LIN {X 0,Y 205.267,Z 502.12,A -85,B 0,C 180,E1 -21304.12,E2 -21304.12} C_VEL
LIN {X 0,Y 202.295,Z 509.063,A -85,B 0,C 180,E1 -21307.536,E2 -21307.536} C_VEL
LIN {X 0,Y 199.763,Z 515.879,A -85,B 0,C 180,E1 -21311.788,E2 -21311.788} C_VEL
LIN {X 0,Y 198.325,Z 520.575,A -85,B 0,C 180,E1 -21315.64,E2 -21315.64} C_VEL
LIN {X 0,Y 197.677,Z 524.301,A -85,B 0,C 180,E1 -21319.763,E2 -21319.763} C_VEL
LIN {X 0,Y 197.879,Z 526.838,A -85,B 0,C 180,E1 -21323.967,E2 -21323.967} C_VEL
LIN {X 0,Y 198.163,Z 528.073,A -85,B 0,C 180,E1 -21327.97,E2 -21327.97} C_VEL
LIN {X 0,Y 198.486,Z 528.261,A -85,B 0,C 180,E1 -21330.003,E2 -21330.003} C_VEL
LIN {X 0,Y 198.017,Z 527.58,A -85,B 0,C 180,E1 -21334.073,E2 -21334.073} C_VEL
LIN {X 0,Y 197.928,Z 526.77,A -85,B 0,C 180,E1 -21336.164,E2 -21336.164} C_VEL
LIN {X 0,Y 197.717,Z 524.267,A -85,B 0,C 180,E1 -21340.24,E2 -21340.24} C_VEL
LIN {X 0,Y 198.347,Z 520.514,A -85,B 0,C 180,E1 -21344.363,E2 -21344.363} C_VEL
LIN {X 0,Y 199.847,Z 515.452,A -85,B 0,C 180,E1 -21348.454,E2 -21348.454} C_VEL
LIN {X 0,Y 202.319,Z 508.963,A -85,B 0,C 180,E1 -21352.467,E2 -21352.467} C_VEL
LIN {X 0,Y 205.735,Z 500.856,A -85,B 0,C 180,E1 -21356.367,E2 -21356.367} C_VEL
LIN {X 0,Y 208.882,Z 493.891,A -85,B 0,C 180,E1 -21359.202,E2 -21359.202} C_VEL
LIN {X 0,Y 214.362,Z 488.856,A -85,B 0,C 180,E1 -21362.752,E2 -21362.752} C_VEL
LIN {X 0,Y 222.751,Z 481.086,A -85,B 0,C 180,E1 -21366.834,E2 -21366.834} C_VEL
LIN {X 0,Y 228.645,Z 475.569,A -85,B 0,C 180,E1 -21369.061,E2 -21369.061} C_VEL
LIN {X 0,Y 239.611,Z 464.861,A -85,B 0,C 180,E1 -21372.426,E2 -21372.426} C_VEL
LIN {X 0,Y 250.645,Z 453.222,A -85,B 0,C 180,E1 -21375.075,E2 -21375.075} C_VEL
LIN {X 0,Y 261.321,Z 440.945,A -85,B 0,C 180,E1 -21377.129,E2 -21377.129} C_VEL
LIN {X 0,Y 269.925,Z 430.113,A -85,B 0,C 180,E1 -21378.468,E2 -21378.468} C_VEL
LIN {X 0,Y 275.364,Z 422.771,A -85,B 0,C 180,E1 -21379.23,E2 -21379.23} C_VEL
LIN {X 0,Y 276.293,Z 421.354,A -85,B 0,C 180,E1 -21379.579,E2 -21379.579} C_VEL
LIN {X 0,Y 267.377,Z 431.541,A -85,B 0,C 180,E1 -21381.372,E2 -21381.372} C_VEL
LIN {X 0,Y 257.679,Z 441.222,A -85,B 0,C 180,E1 -21383.615,E2 -21383.615} C_VEL
LIN {X 0,Y 249.699,Z 448.11,A -85,B 0,C 180,E1 -21385.742,E2 -21385.742} C_VEL
LIN {X 0,Y 241.223,Z 454.408,A -85,B 0,C 180,E1 -21388.37,E2 -21388.37} C_VEL
LIN {X 0,Y 233.351,Z 459.281,A -85,B 0,C 180,E1 -21391.192,E2 -21391.192} C_VEL
LIN {X 0,Y 226.141,Z 462.776,A -85,B 0,C 180,E1 -21394.209,E2 -21394.209} C_VEL
LIN {X 0,Y 219.797,Z 464.844,A -85,B 0,C 180,E1 -21397.437,E2 -21397.437} C_VEL
LIN {X 0,Y 214.14,Z 465.558,A -85,B 0,C 180,E1 -21400.841,E2 -21400.841} C_VEL
LIN {X 0,Y 209.476,Z 464.862,A -85,B 0,C 180,E1 -21404.431,E2 -21404.431} C_VEL
LIN {X 0,Y 205.6,Z 462.774,A -85,B 0,C 180,E1 -21408.165,E2 -21408.165} C_VEL
LIN {X 0,Y 202.968,Z 459.202,A -85,B 0,C 180,E1 -21412.039,E2 -21412.039} C_VEL
LIN {X 0,Y 200.986,Z 454.078,A -85,B 0,C 180,E1 -21415.99,E2 -21415.99} C_VEL
LIN {X 0,Y 199.711,Z 447.24,A -85,B 0,C 180,E1 -21420,E2 -21420} C_VEL
LIN {X 0,Y 199.428,Z 440.84,A -85,B 0,C 180,E1 -21423.03,E2 -21423.03} C_VEL
LIN {X 0,Y 199.398,Z 433.173,A -85,B 0,C 180,E1 -21426.07,E2 -21426.07} C_VEL
LIN {X 0,Y 199.905,Z 424.141,A -85,B 0,C 180,E1 -21429.076,E2 -21429.076} C_VEL
LIN {X 0,Y 200.647,Z 413.012,A -85,B 0,C 180,E1 -21432.132,E2 -21432.132} C_VEL
LIN {X 0,Y 201.556,Z 400.828,A -85,B 0,C 180,E1 -21434.902,E2 -21434.902} C_VEL
LIN {X 0,Y 202.642,Z 387.299,A -85,B 0,C 180,E1 -21437.406,E2 -21437.406} C_VEL
LIN {X 0,Y 203.727,Z 374.15,A -85,B 0,C 180,E1 -21439.393,E2 -21439.393} C_VEL
LIN {X 0,Y 204.695,Z 359.774,A -85,B 0,C 180,E1 -21441.132,E2 -21441.132} C_VEL
LIN {X 0,Y 205.639,Z 343.824,A -85,B 0,C 180,E1 -21442.623,E2 -21442.623} C_VEL
LIN {X 0,Y 206.657,Z 321.429,A -85,B 0,C 180,E1 -21444.086,E2 -21444.086} C_VEL
LIN {X 0,Y 211.562,Z 242.2,A -85,B 0,C 180,E1 -21448.698,E2 -21448.698} C_VEL
LIN {X 0,Y 211.534,Z 241.628,A -85,B 0,C 180,E1 -21448.781,E2 -21448.781} C_VEL
LIN {X 0,Y 213.23,Z 241.827,A -85,B 0,C 180,E1 -21449.63,E2 -21449.63} C_VEL
LIN {X 0,Y 214.627,Z 239.56,A -85,B 0,C 180,E1 -21450.143,E2 -21450.143} C_VEL
LIN {X 0,Y 216.77,Z 233.61,A -85,B 0,C 180,E1 -21450.741,E2 -21450.741} C_VEL
LIN {X 0,Y 218.364,Z 227.891,A -85,B 0,C 180,E1 -21451.09,E2 -21451.09} C_VEL
LIN {X 0,Y 220.497,Z 225.426,A -85,B 0,C 180,E1 -21451.864,E2 -21451.864} C_VEL
LIN {X 0,Y 222.215,Z 222.209,A -85,B 0,C 180,E1 -21452.39,E2 -21452.39} C_VEL
LIN {X 0,Y 224.392,Z 221.596,A -85,B 0,C 180,E1 -21453.237,E2 -21453.237} C_VEL
LIN {X 0,Y 228.278,Z 221.524,A -85,B 0,C 180,E1 -21454.72,E2 -21454.72} C_VEL
LIN {X 0,Y 231.326,Z 221.102,A -85,B 0,C 180,E1 -21455.792,E2 -21455.792} C_VEL
LIN {X 0,Y 232.183,Z 221.454,A -85,B 0,C 180,E1 -21456.108,E2 -21456.108} C_VEL
LIN {X 0,Y 237.875,Z 230.482,A -85,B 0,C 180,E1 -21458.416,E2 -21458.416} C_VEL
LIN {X 0,Y 244.244,Z 241.683,A -85,B 0,C 180,E1 -21460.797,E2 -21460.797} C_VEL
LIN {X 0,Y 250.045,Z 253.287,A -85,B 0,C 180,E1 -21462.827,E2 -21462.827} C_VEL
LIN {X 0,Y 243.977,Z 351.523,A -85,B 0,C 180,E1 -21465.471,E2 -21465.471} C_VEL
LIN {X 0,Y 242.422,Z 366.589,A -85,B 0,C 180,E1 -21466.149,E2 -21466.149} C_VEL
LIN {X 0,Y 240.345,Z 380.819,A -85,B 0,C 180,E1 -21467.092,E2 -21467.092} C_VEL
LIN {X 0,Y 237.764,Z 394.532,A -85,B 0,C 180,E1 -21468.31,E2 -21468.31} C_VEL
LIN {X 0,Y 234.321,Z 408.371,A -85,B 0,C 180,E1 -21469.843,E2 -21469.843} C_VEL
LIN {X 0,Y 230.62,Z 420.997,A -85,B 0,C 180,E1 -21471.615,E2 -21471.615} C_VEL
LIN {X 0,Y 226.485,Z 432.68,A -85,B 0,C 180,E1 -21473.595,E2 -21473.595} C_VEL
LIN {X 0,Y 222.424,Z 443.47,A -85,B 0,C 180,E1 -21475.883,E2 -21475.883} C_VEL
LIN {X 0,Y 218.441,Z 453.372,A -85,B 0,C 180,E1 -21478.476,E2 -21478.476} C_VEL
LIN {X 0,Y 213.958,Z 463.052,A -85,B 0,C 180,E1 -21481.554,E2 -21481.554} C_VEL
LIN {X 0,Y 209.892,Z 471.448,A -85,B 0,C 180,E1 -21484.916,E2 -21484.916} C_VEL
LIN {X 0,Y 206.815,Z 477.669,A -85,B 0,C 180,E1 -21488.047,E2 -21488.047} C_VEL
LIN {X 0,Y 203.821,Z 483.766,A -85,B 0,C 180,E1 -21491.918,E2 -21491.918} C_VEL
LIN {X 0,Y 201.497,Z 488.471,A -85,B 0,C 180,E1 -21495.866,E2 -21495.866} C_VEL
LIN {X 0,Y 199.865,Z 491.947,A -85,B 0,C 180,E1 -21499.928,E2 -21499.928} C_VEL
LIN {X 0,Y 198.859,Z 494.17,A -85,B 0,C 180,E1 -21503.911,E2 -21503.911} C_VEL
LIN {X 0,Y 198.504,Z 495.303,A -85,B 0,C 180,E1 -21507.968,E2 -21507.968} C_VEL
LIN {X 0,Y 198.503,Z 495.314,A -85,B 0,C 180,E1 -21512.026,E2 -21512.026} C_VEL
LIN {X 0,Y 198.844,Z 494.224,A -85,B 0,C 180,E1 -21516.084,E2 -21516.084} C_VEL
LIN {X 0,Y 199.896,Z 492.006,A -85,B 0,C 180,E1 -21520.122,E2 -21520.122} C_VEL
LIN {X 0,Y 201.475,Z 488.625,A -85,B 0,C 180,E1 -21524.131,E2 -21524.131} C_VEL
LIN {X 0,Y 203.746,Z 483.977,A -85,B 0,C 180,E1 -21528.083,E2 -21528.083} C_VEL
LIN {X 0,Y 206.75,Z 477.926,A -85,B 0,C 180,E1 -21531.955,E2 -21531.955} C_VEL
LIN {X 0,Y 210.505,Z 470.295,A -85,B 0,C 180,E1 -21535.72,E2 -21535.72} C_VEL
LIN {X 0,Y 214.482,Z 462.127,A -85,B 0,C 180,E1 -21538.899,E2 -21538.899} C_VEL
LIN {X 0,Y 218.318,Z 453.818,A -85,B 0,C 180,E1 -21541.538,E2 -21541.538} C_VEL
LIN {X 0,Y 223.004,Z 442.178,A -85,B 0,C 180,E1 -21544.557,E2 -21544.557} C_VEL
LIN {X 0,Y 227.205,Z 431.186,A -85,B 0,C 180,E1 -21546.818,E2 -21546.818} C_VEL
LIN {X 0,Y 231.291,Z 419.223,A -85,B 0,C 180,E1 -21548.804,E2 -21548.804} C_VEL
LIN {X 0,Y 235.067,Z 406.182,A -85,B 0,C 180,E1 -21550.559,E2 -21550.559} C_VEL
LIN {X 0,Y 238.502,Z 391.783,A -85,B 0,C 180,E1 -21552.093,E2 -21552.093} C_VEL
LIN {X 0,Y 241.052,Z 377.556,A -85,B 0,C 180,E1 -21553.284,E2 -21553.284} C_VEL
LIN {X 0,Y 243.012,Z 363.087,A -85,B 0,C 180,E1 -21554.167,E2 -21554.167} C_VEL
LIN {X 0,Y 244.401,Z 347.756,A -85,B 0,C 180,E1 -21554.787,E2 -21554.787} C_VEL
LIN {X 0,Y 250.189,Z 254.587,A -85,B 0,C 180,E1 -21557.244,E2 -21557.244} C_VEL
LIN {X 0,Y 250.038,Z 253.089,A -85,B 0,C 180,E1 -21557.345,E2 -21557.345} C_VEL
LIN {X 0,Y 243.731,Z 240.661,A -85,B 0,C 180,E1 -21559.562,E2 -21559.562} C_VEL
LIN {X 0,Y 237.84,Z 230.373,A -85,B 0,C 180,E1 -21561.779,E2 -21561.779} C_VEL
LIN {X 0,Y 230.643,Z 218.967,A -85,B 0,C 180,E1 -21564.756,E2 -21564.756} C_VEL
LIN {X 0,Y 224.207,Z 209.923,A -85,B 0,C 180,E1 -21567.733,E2 -21567.733} C_VEL
LIN {X 0,Y 221.031,Z 205.72,A -85,B 0,C 180,E1 -21569.35,E2 -21569.35} C_VEL
LIN {X 0,Y 215.034,Z 198.081,A -85,B 0,C 180,E1 -21572.77,E2 -21572.77} C_VEL
LIN {X 0,Y 211.661,Z 194.11,A -85,B 0,C 180,E1 -21574.954,E2 -21574.954} C_VEL
LIN {X 0,Y 206.906,Z 188.668,A -85,B 0,C 180,E1 -21578.518,E2 -21578.518} C_VEL
LIN {X 0,Y 204.047,Z 184.332,A -85,B 0,C 180,E1 -21582.976,E2 -21582.976} C_VEL
LIN {X 0,Y 203.68,Z 183.173,A -85,B 0,C 180,E1 -21583.976,E2 -21583.976} C_VEL
LIN {X 0,Y 200.533,Z 178.839,A -85,B 0,C 180,E1 -21591.941,E2 -21591.941} C_VEL
LIN {X 0,Y 200.035,Z 177.181,A -85,B 0,C 180,E1 -21595.97,E2 -21595.97} C_VEL
LIN {X 0,Y 200.473,Z 177.102,A -85,B 0,C 180,E1 -21600,E2 -21600} C_VEL
LIN {X 0,Y 200.144,Z 177.263,A -85,B 0,C 180,E1 -21603.019,E2 -21603.019} C_VEL
LIN {X 0,Y 201.554,Z 180.696,A -85,B 0,C 180,E1 -21609.479,E2 -21609.479} C_VEL
LIN {X 0,Y 202.043,Z 182.351,A -85,B 0,C 180,E1 -21611.083,E2 -21611.083} C_VEL
LIN {X 0,Y 202.303,Z 186.976,A -85,B 0,C 180,E1 -21613.573,E2 -21613.573} C_VEL
LIN {X 0,Y 202.846,Z 191.885,A -85,B 0,C 180,E1 -21616.039,E2 -21616.039} C_VEL
LIN {X 0,Y 203.809,Z 193.97,A -85,B 0,C 180,E1 -21617.592,E2 -21617.592} C_VEL
LIN {X 0,Y 208.306,Z 200.489,A -85,B 0,C 180,E1 -21622.622,E2 -21622.622} C_VEL
LIN {X 0,Y 212.381,Z 205.711,A -85,B 0,C 180,E1 -21625.479,E2 -21625.479} C_VEL
LIN {X 0,Y 215.855,Z 210.205,A -85,B 0,C 180,E1 -21627.629,E2 -21627.629} C_VEL
LIN {X 0,Y 220.293,Z 216.142,A -85,B 0,C 180,E1 -21630.097,E2 -21630.097} C_VEL
LIN {X 0,Y 226.822,Z 225.523,A -85,B 0,C 180,E1 -21633.314,E2 -21633.314} C_VEL
LIN {X 0,Y 230.886,Z 232,A -85,B 0,C 180,E1 -21635.134,E2 -21635.134} C_VEL
LIN {X 0,Y 236.073,Z 246.149,A -85,B 0,C 180,E1 -21637.547,E2 -21637.547} C_VEL
LIN {X 0,Y 241.184,Z 260.671,A -85,B 0,C 180,E1 -21639.736,E2 -21639.736} C_VEL
LIN {X 0,Y 242.647,Z 292.092,A -85,B 0,C 180,E1 -21641.521,E2 -21641.521} C_VEL
LIN {X 0,Y 236.96,Z 380.814,A -85,B 0,C 180,E1 -21643.936,E2 -21643.936} C_VEL
LIN {X 0,Y 234.922,Z 396.302,A -85,B 0,C 180,E1 -21644.575,E2 -21644.575} C_VEL
LIN {X 0,Y 232.241,Z 410.574,A -85,B 0,C 180,E1 -21645.441,E2 -21645.441} C_VEL
LIN {X 0,Y 228.783,Z 424.674,A -85,B 0,C 180,E1 -21646.584,E2 -21646.584} C_VEL
LIN {X 0,Y 224.728,Z 438.446,A -85,B 0,C 180,E1 -21648.055,E2 -21648.055} C_VEL
LIN {X 0,Y 220.379,Z 451.105,A -85,B 0,C 180,E1 -21649.779,E2 -21649.779} C_VEL
LIN {X 0,Y 215.524,Z 463.933,A -85,B 0,C 180,E1 -21652.016,E2 -21652.016} C_VEL
LIN {X 0,Y 210.925,Z 474.673,A -85,B 0,C 180,E1 -21654.335,E2 -21654.335} C_VEL
LIN {X 0,Y 206.54,Z 484.646,A -85,B 0,C 180,E1 -21657.017,E2 -21657.017} C_VEL
LIN {X 0,Y 201.94,Z 494.543,A -85,B 0,C 180,E1 -21660.33,E2 -21660.33} C_VEL
LIN {X 0,Y 198.325,Z 502.592,A -85,B 0,C 180,E1 -21663.71,E2 -21663.71} C_VEL
LIN {X 0,Y 194.879,Z 510.235,A -85,B 0,C 180,E1 -21667.752,E2 -21667.752} C_VEL
LIN {X 0,Y 192.765,Z 515.719,A -85,B 0,C 180,E1 -21671.429,E2 -21671.429} C_VEL
LIN {X 0,Y 191.085,Z 521.064,A -85,B 0,C 180,E1 -21676.171,E2 -21676.171} C_VEL
LIN {X 0,Y 190.622,Z 523.709,A -85,B 0,C 180,E1 -21679.38,E2 -21679.38} C_VEL
LIN {X 0,Y 190.796,Z 526.359,A -85,B 0,C 180,E1 -21684.013,E2 -21684.013} C_VEL
LIN {X 0,Y 191.069,Z 527.486,A -85,B 0,C 180,E1 -21687.895,E2 -21687.895} C_VEL
LIN {X 0,Y 191.407,Z 527.675,A -85,B 0,C 180,E1 -21690.003,E2 -21690.003} C_VEL
LIN {X 0,Y 190.943,Z 526.994,A -85,B 0,C 180,E1 -21694.224,E2 -21694.224} C_VEL
LIN {X 0,Y 190.835,Z 526.199,A -85,B 0,C 180,E1 -21696.346,E2 -21696.346} C_VEL
LIN {X 0,Y 190.658,Z 523.674,A -85,B 0,C 180,E1 -21700.624,E2 -21700.624} C_VEL
LIN {X 0,Y 191.385,Z 519.92,A -85,B 0,C 180,E1 -21704.898,E2 -21704.898} C_VEL
LIN {X 0,Y 193.025,Z 514.856,A -85,B 0,C 180,E1 -21709.131,E2 -21709.131} C_VEL
LIN {X 0,Y 195.674,Z 508.367,A -85,B 0,C 180,E1 -21713.274,E2 -21713.274} C_VEL
LIN {X 0,Y 199.314,Z 500.262,A -85,B 0,C 180,E1 -21717.286,E2 -21717.286} C_VEL
LIN {X 0,Y 202.236,Z 493.928,A -85,B 0,C 180,E1 -21719.887,E2 -21719.887} C_VEL
LIN {X 0,Y 208.409,Z 488.894,A -85,B 0,C 180,E1 -21723.811,E2 -21723.811} C_VEL
LIN {X 0,Y 217.126,Z 481.673,A -85,B 0,C 180,E1 -21727.954,E2 -21727.954} C_VEL
LIN {X 0,Y 223.225,Z 476.54,A -85,B 0,C 180,E1 -21730.2,E2 -21730.2} C_VEL
LIN {X 0,Y 233.391,Z 467.62,A -85,B 0,C 180,E1 -21733.243,E2 -21733.243} C_VEL
LIN {X 0,Y 243.294,Z 458.29,A -85,B 0,C 180,E1 -21735.642,E2 -21735.642} C_VEL
LIN {X 0,Y 252.595,Z 448.843,A -85,B 0,C 180,E1 -21737.506,E2 -21737.506} C_VEL
LIN {X 0,Y 262.509,Z 437.915,A -85,B 0,C 180,E1 -21739.143,E2 -21739.143} C_VEL
LIN {X 0,Y 265.313,Z 434.636,A -85,B 0,C 180,E1 -21739.549,E2 -21739.549} C_VEL
LIN {X 0,Y 266.15,Z 433.507,A -85,B 0,C 180,E1 -21739.875,E2 -21739.875} C_VEL
LIN {X 0,Y 256.421,Z 442.613,A -85,B 0,C 180,E1 -21741.926,E2 -21741.926} C_VEL
LIN {X 0,Y 246.802,Z 450.333,A -85,B 0,C 180,E1 -21744.284,E2 -21744.284} C_VEL
LIN {X 0,Y 237.868,Z 456.432,A -85,B 0,C 180,E1 -21746.866,E2 -21746.866} C_VEL
LIN {X 0,Y 231.565,Z 460.083,A -85,B 0,C 180,E1 -21748.939,E2 -21748.939} C_VEL
LIN {X 0,Y 223.736,Z 463.733,A -85,B 0,C 180,E1 -21751.889,E2 -21751.889} C_VEL
LIN {X 0,Y 216.709,Z 466.035,A -85,B 0,C 180,E1 -21755.065,E2 -21755.065} C_VEL
LIN {X 0,Y 210.451,Z 467.023,A -85,B 0,C 180,E1 -21758.448,E2 -21758.448} C_VEL
LIN {X 0,Y 205.01,Z 466.669,A -85,B 0,C 180,E1 -21762.029,E2 -21762.029} C_VEL
LIN {X 0,Y 200.544,Z 464.901,A -85,B 0,C 180,E1 -21765.8,E2 -21765.8} C_VEL
LIN {X 0,Y 197.186,Z 461.665,A -85,B 0,C 180,E1 -21769.735,E2 -21769.735} C_VEL
LIN {X 0,Y 195.338,Z 458.307,A -85,B 0,C 180,E1 -21772.766,E2 -21772.766} C_VEL
LIN {X 0,Y 193.494,Z 452.366,A -85,B 0,C 180,E1 -21776.877,E2 -21776.877} C_VEL
LIN {X 0,Y 192.586,Z 445.746,A -85,B 0,C 180,E1 -21780.523,E2 -21780.523} C_VEL
LIN {X 0,Y 192.376,Z 437.587,A -85,B 0,C 180,E1 -21784.19,E2 -21784.19} C_VEL
LIN {X 0,Y 192.555,Z 429.085,A -85,B 0,C 180,E1 -21787.34,E2 -21787.34} C_VEL
LIN {X 0,Y 192.977,Z 420.635,A -85,B 0,C 180,E1 -21789.995,E2 -21789.995} C_VEL
LIN {X 0,Y 193.846,Z 408.825,A -85,B 0,C 180,E1 -21793.097,E2 -21793.097} C_VEL
LIN {X 0,Y 194.792,Z 396.892,A -85,B 0,C 180,E1 -21795.7,E2 -21795.7} C_VEL
LIN {X 0,Y 195.841,Z 383.889,A -85,B 0,C 180,E1 -21798.03,E2 -21798.03} C_VEL
LIN {X 0,Y 197.027,Z 369.847,A -85,B 0,C 180,E1 -21800.08,E2 -21800.08} C_VEL
LIN {X 0,Y 197.929,Z 355.377,A -85,B 0,C 180,E1 -21801.754,E2 -21801.754} C_VEL
LIN {X 0,Y 198.812,Z 339.04,A -85,B 0,C 180,E1 -21803.183,E2 -21803.183} C_VEL
LIN {X 0,Y 201.705,Z 284.183,A -85,B 0,C 180,E1 -21806.654,E2 -21806.654} C_VEL
LIN {X 0,Y 201.967,Z 285.337,A -85,B 0,C 180,E1 -21806.896,E2 -21806.896} C_VEL
LIN {X 0,Y 202.861,Z 285.273,A -85,B 0,C 180,E1 -21807.395,E2 -21807.395} C_VEL
LIN {X 0,Y 204.303,Z 282.16,A -85,B 0,C 180,E1 -21807.95,E2 -21807.95} C_VEL
LIN {X 0,Y 207.227,Z 273.064,A -85,B 0,C 180,E1 -21808.823,E2 -21808.823} C_VEL
LIN {X 0,Y 211.208,Z 258.049,A -85,B 0,C 180,E1 -21809.757,E2 -21809.757} C_VEL
LIN {X 0,Y 213.505,Z 248.555,A -85,B 0,C 180,E1 -21810.213,E2 -21810.213} C_VEL
LIN {X 0,Y 215.285,Z 246.777,A -85,B 0,C 180,E1 -21810.918,E2 -21810.918} C_VEL
LIN {X 0,Y 217.271,Z 243.285,A -85,B 0,C 180,E1 -21811.58,E2 -21811.58} C_VEL
LIN {X 0,Y 219.622,Z 237.131,A -85,B 0,C 180,E1 -21812.209,E2 -21812.209} C_VEL
LIN {X 0,Y 221.028,Z 232.529,A -85,B 0,C 180,E1 -21812.518,E2 -21812.518} C_VEL
LIN {X 0,Y 223.655,Z 228.769,A -85,B 0,C 180,E1 -21813.361,E2 -21813.361} C_VEL
LIN {X 0,Y 229.09,Z 228.308,A -85,B 0,C 180,E1 -21815.384,E2 -21815.384} C_VEL
LIN {X 0,Y 229.972,Z 228.318,A -85,B 0,C 180,E1 -21815.698,E2 -21815.698} C_VEL
LIN {X 0,Y 236.628,Z 239.388,A -85,B 0,C 180,E1 -21818.46,E2 -21818.46} C_VEL
LIN {X 0,Y 243.014,Z 251.542,A -85,B 0,C 180,E1 -21820.897,E2 -21820.897} C_VEL
LIN {X 0,Y 245.146,Z 255.943,A -85,B 0,C 180,E1 -21821.671,E2 -21821.671} C_VEL
LIN {X 0,Y 238.88,Z 353.426,A -85,B 0,C 180,E1 -21824.331,E2 -21824.331} C_VEL
LIN {X 0,Y 237.177,Z 368.658,A -85,B 0,C 180,E1 -21825.05,E2 -21825.05} C_VEL
LIN {X 0,Y 234.992,Z 382.565,A -85,B 0,C 180,E1 -21826.008,E2 -21826.008} C_VEL
LIN {X 0,Y 232.071,Z 397.023,A -85,B 0,C 180,E1 -21827.341,E2 -21827.341} C_VEL
LIN {X 0,Y 228.971,Z 408.944,A -85,B 0,C 180,E1 -21828.704,E2 -21828.704} C_VEL
LIN {X 0,Y 225.121,Z 421.574,A -85,B 0,C 180,E1 -21830.497,E2 -21830.497} C_VEL
LIN {X 0,Y 220.83,Z 433.259,A -85,B 0,C 180,E1 -21832.505,E2 -21832.505} C_VEL
LIN {X 0,Y 216.602,Z 444.051,A -85,B 0,C 180,E1 -21834.833,E2 -21834.833} C_VEL
LIN {X 0,Y 212.435,Z 453.955,A -85,B 0,C 180,E1 -21837.477,E2 -21837.477} C_VEL
LIN {X 0,Y 207.747,Z 463.637,A -85,B 0,C 180,E1 -21840.622,E2 -21840.622} C_VEL
LIN {X 0,Y 203.404,Z 472.226,A -85,B 0,C 180,E1 -21844.161,E2 -21844.161} C_VEL
LIN {X 0,Y 200.27,Z 478.254,A -85,B 0,C 180,E1 -21847.29,E2 -21847.29} C_VEL
LIN {X 0,Y 197.077,Z 484.353,A -85,B 0,C 180,E1 -21851.277,E2 -21851.277} C_VEL
LIN {X 0,Y 194.638,Z 489.057,A -85,B 0,C 180,E1 -21855.357,E2 -21855.357} C_VEL
LIN {X 0,Y 192.844,Z 492.648,A -85,B 0,C 180,E1 -21859.734,E2 -21859.734} C_VEL
LIN {X 0,Y 191.82,Z 494.755,A -85,B 0,C 180,E1 -21863.687,E2 -21863.687} C_VEL
LIN {X 0,Y 191.446,Z 495.887,A -85,B 0,C 180,E1 -21867.894,E2 -21867.894} C_VEL
LIN {X 0,Y 191.445,Z 495.897,A -85,B 0,C 180,E1 -21872.101,E2 -21872.101} C_VEL
LIN {X 0,Y 191.806,Z 494.808,A -85,B 0,C 180,E1 -21876.308,E2 -21876.308} C_VEL
LIN {X 0,Y 192.941,Z 492.589,A -85,B 0,C 180,E1 -21880.491,E2 -21880.491} C_VEL
LIN {X 0,Y 194.617,Z 489.209,A -85,B 0,C 180,E1 -21884.639,E2 -21884.639} C_VEL
LIN {X 0,Y 197.004,Z 484.562,A -85,B 0,C 180,E1 -21888.725,E2 -21888.725} C_VEL
LIN {X 0,Y 200.2,Z 478.508,A -85,B 0,C 180,E1 -21892.712,E2 -21892.712} C_VEL
LIN {X 0,Y 204.152,Z 470.876,A -85,B 0,C 180,E1 -21896.582,E2 -21896.582} C_VEL
LIN {X 0,Y 208.299,Z 462.708,A -85,B 0,C 180,E1 -21899.842,E2 -21899.842} C_VEL
LIN {X 0,Y 212.321,Z 454.396,A -85,B 0,C 180,E1 -21902.537,E2 -21902.537} C_VEL
LIN {X 0,Y 216.475,Z 444.556,A -85,B 0,C 180,E1 -21905.185,E2 -21905.185} C_VEL
LIN {X 0,Y 220.741,Z 433.864,A -85,B 0,C 180,E1 -21907.507,E2 -21907.507} C_VEL
LIN {X 0,Y 224.971,Z 422.304,A -85,B 0,C 180,E1 -21909.528,E2 -21909.528} C_VEL
LIN {X 0,Y 228.841,Z 409.817,A -85,B 0,C 180,E1 -21911.319,E2 -21911.319} C_VEL
LIN {X 0,Y 232.42,Z 396.19,A -85,B 0,C 180,E1 -21912.869,E2 -21912.869} C_VEL
LIN {X 0,Y 235.412,Z 381.089,A -85,B 0,C 180,E1 -21914.234,E2 -21914.234} C_VEL
LIN {X 0,Y 237.671,Z 366.217,A -85,B 0,C 180,E1 -21915.206,E2 -21915.206} C_VEL
LIN {X 0,Y 239.238,Z 351.009,A -85,B 0,C 180,E1 -21915.877,E2 -21915.877} C_VEL
LIN {X 0,Y 245.297,Z 256.104,A -85,B 0,C 180,E1 -21918.448,E2 -21918.448} C_VEL
LIN {X 0,Y 239.39,Z 244.378,A -85,B 0,C 180,E1 -21920.643,E2 -21920.643} C_VEL
LIN {X 0,Y 233.393,Z 233.803,A -85,B 0,C 180,E1 -21923.037,E2 -21923.037} C_VEL
LIN {X 0,Y 227.065,Z 223.766,A -85,B 0,C 180,E1 -21925.808,E2 -21925.808} C_VEL
LIN {X 0,Y 221.739,Z 216.035,A -85,B 0,C 180,E1 -21928.398,E2 -21928.398} C_VEL
LIN {X 0,Y 216.747,Z 209.284,A -85,B 0,C 180,E1 -21931.112,E2 -21931.112} C_VEL
LIN {X 0,Y 212.619,Z 204.089,A -85,B 0,C 180,E1 -21933.63,E2 -21933.63} C_VEL
LIN {X 0,Y 209.554,Z 200.266,A -85,B 0,C 180,E1 -21935.726,E2 -21935.726} C_VEL
LIN {X 0,Y 205.285,Z 195.346,A -85,B 0,C 180,E1 -21939.063,E2 -21939.063} C_VEL
LIN {X 0,Y 200.595,Z 190.035,A -85,B 0,C 180,E1 -21943.722,E2 -21943.722} C_VEL
LIN {X 0,Y 199.629,Z 188.534,A -85,B 0,C 180,E1 -21945.733,E2 -21945.733} C_VEL
LIN {X 0,Y 197.255,Z 184.511,A -85,B 0,C 180,E1 -21953.864,E2 -21953.864} C_VEL
LIN {X 0,Y 197.075,Z 183.547,A -85,B 0,C 180,E1 -21956.829,E2 -21956.829} C_VEL
LIN {X 0,Y 197.113,Z 183.339,A -85,B 0,C 180,E1 -21960,E2 -21960} C_VEL
LIN {X 0,Y 197.301,Z 183.555,A -85,B 0,C 180,E1 -21962.041,E2 -21962.041} C_VEL
LIN {X 0,Y 200.272,Z 188.836,A -85,B 0,C 180,E1 -21972.155,E2 -21972.155} C_VEL
LIN {X 0,Y 203.809,Z 193.97,A -85,B 0,C 180,E1 -21977.592,E2 -21977.592} C_VEL
LIN {X 0,Y 204.985,Z 196.202,A -85,B 0,C 180,E1 -21979.08,E2 -21979.08} C_VEL
LIN {X 0,Y 205.976,Z 199.486,A -85,B 0,C 180,E1 -21980.429,E2 -21980.429} C_VEL
LIN {X 0,Y 208.951,Z 209.62,A -85,B 0,C 180,E1 -21983.769,E2 -21983.769} C_VEL
LIN {X 0,Y 210.105,Z 211.719,A -85,B 0,C 180,E1 -21984.65,E2 -21984.65} C_VEL
LIN {X 0,Y 213.575,Z 216.329,A -85,B 0,C 180,E1 -21986.902,E2 -21986.902} C_VEL
LIN {X 0,Y 217.621,Z 221.919,A -85,B 0,C 180,E1 -21989.261,E2 -21989.261} C_VEL
LIN {X 0,Y 223.053,Z 229.913,A -85,B 0,C 180,E1 -21992.094,E2 -21992.094} C_VEL
LIN {X 0,Y 227.557,Z 237.177,A -85,B 0,C 180,E1 -21994.227,E2 -21994.227} C_VEL
LIN {X 0,Y 233.642,Z 254.438,A -85,B 0,C 180,E1 -21997.187,E2 -21997.187} C_VEL
LIN {X 0,Y 236.76,Z 263.883,A -85,B 0,C 180,E1 -21998.602,E2 -21998.602} C_VEL
LIN {X 0,Y 237.895,Z 293.498,A -85,B 0,C 180,E1 -22000.296,E2 -22000.296} C_VEL
LIN {X 0,Y 232.077,Z 380.328,A -85,B 0,C 180,E1 -22002.67,E2 -22002.67} C_VEL
LIN {X 0,Y 229.999,Z 395.774,A -85,B 0,C 180,E1 -22003.316,E2 -22003.316} C_VEL
LIN {X 0,Y 226.95,Z 411.303,A -85,B 0,C 180,E1 -22004.269,E2 -22004.269} C_VEL
LIN {X 0,Y 223.155,Z 426.079,A -85,B 0,C 180,E1 -22005.518,E2 -22005.518} C_VEL
LIN {X 0,Y 218.97,Z 439.45,A -85,B 0,C 180,E1 -22007.001,E2 -22007.001} C_VEL
LIN {X 0,Y 214.491,Z 451.818,A -85,B 0,C 180,E1 -22008.748,E2 -22008.748} C_VEL
LIN {X 0,Y 209.915,Z 463.351,A -85,B 0,C 180,E1 -22010.81,E2 -22010.81} C_VEL
LIN {X 0,Y 205.156,Z 474.09,A -85,B 0,C 180,E1 -22013.17,E2 -22013.17} C_VEL
LIN {X 0,Y 200.531,Z 484.057,A -85,B 0,C 180,E1 -22015.896,E2 -22015.896} C_VEL
LIN {X 0,Y 195.806,Z 493.829,A -85,B 0,C 180,E1 -22019.242,E2 -22019.242} C_VEL
LIN {X 0,Y 191.883,Z 501.999,A -85,B 0,C 180,E1 -22022.756,E2 -22022.756} C_VEL
LIN {X 0,Y 188.241,Z 509.643,A -85,B 0,C 180,E1 -22026.923,E2 -22026.923} C_VEL
LIN {X 0,Y 185.813,Z 515.484,A -85,B 0,C 180,E1 -22031.009,E2 -22031.009} C_VEL
LIN {X 0,Y 184.119,Z 520.471,A -85,B 0,C 180,E1 -22035.637,E2 -22035.637} C_VEL
LIN {X 0,Y 183.551,Z 523.115,A -85,B 0,C 180,E1 -22038.966,E2 -22038.966} C_VEL
LIN {X 0,Y 183.714,Z 525.879,A -85,B 0,C 180,E1 -22044.06,E2 -22044.06} C_VEL
LIN {X 0,Y 183.978,Z 526.9,A -85,B 0,C 180,E1 -22047.814,E2 -22047.814} C_VEL
LIN {X 0,Y 184.329,Z 527.091,A -85,B 0,C 180,E1 -22050.003,E2 -22050.003} C_VEL
LIN {X 0,Y 183.869,Z 526.407,A -85,B 0,C 180,E1 -22054.387,E2 -22054.387} C_VEL
LIN {X 0,Y 183.731,Z 525.608,A -85,B 0,C 180,E1 -22056.592,E2 -22056.592} C_VEL
LIN {X 0,Y 183.601,Z 523.08,A -85,B 0,C 180,E1 -22061.037,E2 -22061.037} C_VEL
LIN {X 0,Y 184.443,Z 519.325,A -85,B 0,C 180,E1 -22065.472,E2 -22065.472} C_VEL
LIN {X 0,Y 186.226,Z 514.26,A -85,B 0,C 180,E1 -22069.858,E2 -22069.858} C_VEL
LIN {X 0,Y 189.066,Z 507.771,A -85,B 0,C 180,E1 -22074.138,E2 -22074.138} C_VEL
LIN {X 0,Y 192.957,Z 499.669,A -85,B 0,C 180,E1 -22078.264,E2 -22078.264} C_VEL
LIN {X 0,Y 195.99,Z 493.535,A -85,B 0,C 180,E1 -22080.882,E2 -22080.882} C_VEL
LIN {X 0,Y 202.522,Z 488.858,A -85,B 0,C 180,E1 -22084.934,E2 -22084.934} C_VEL
LIN {X 0,Y 211.592,Z 482.184,A -85,B 0,C 180,E1 -22089.133,E2 -22089.133} C_VEL
LIN {X 0,Y 217.901,Z 477.464,A -85,B 0,C 180,E1 -22091.393,E2 -22091.393} C_VEL
LIN {X 0,Y 229.565,Z 468.135,A -85,B 0,C 180,E1 -22094.762,E2 -22094.762} C_VEL
LIN {X 0,Y 241.183,Z 458.08,A -85,B 0,C 180,E1 -22097.375,E2 -22097.375} C_VEL
LIN {X 0,Y 252.289,Z 447.568,A -85,B 0,C 180,E1 -22099.388,E2 -22099.388} C_VEL
LIN {X 0,Y 255.052,Z 444.811,A -85,B 0,C 180,E1 -22099.83,E2 -22099.83} C_VEL
LIN {X 0,Y 255.27,Z 444.326,A -85,B 0,C 180,E1 -22100.293,E2 -22100.293} C_VEL
LIN {X 0,Y 246.6,Z 450.943,A -85,B 0,C 180,E1 -22102.212,E2 -22102.212} C_VEL
LIN {X 0,Y 237.01,Z 457.207,A -85,B 0,C 180,E1 -22104.674,E2 -22104.674} C_VEL
LIN {X 0,Y 228.08,Z 462.026,A -85,B 0,C 180,E1 -22107.368,E2 -22107.368} C_VEL
LIN {X 0,Y 221.822,Z 464.785,A -85,B 0,C 180,E1 -22109.541,E2 -22109.541} C_VEL
LIN {X 0,Y 214.061,Z 467.285,A -85,B 0,C 180,E1 -22112.636,E2 -22112.636} C_VEL
LIN {X 0,Y 207.186,Z 468.467,A -85,B 0,C 180,E1 -22115.98,E2 -22115.98} C_VEL
LIN {X 0,Y 201.043,Z 468.368,A -85,B 0,C 180,E1 -22119.539,E2 -22119.539} C_VEL
LIN {X 0,Y 195.999,Z 466.88,A -85,B 0,C 180,E1 -22123.33,E2 -22123.33} C_VEL
LIN {X 0,Y 191.81,Z 464.03,A -85,B 0,C 180,E1 -22127.3,E2 -22127.3} C_VEL
LIN {X 0,Y 188.96,Z 459.715,A -85,B 0,C 180,E1 -22131.444,E2 -22131.444} C_VEL
LIN {X 0,Y 187.275,Z 455.453,A -85,B 0,C 180,E1 -22134.617,E2 -22134.617} C_VEL
LIN {X 0,Y 185.994,Z 450.22,A -85,B 0,C 180,E1 -22137.835,E2 -22137.835} C_VEL
LIN {X 0,Y 185.435,Z 442.843,A -85,B 0,C 180,E1 -22141.629,E2 -22141.629} C_VEL
LIN {X 0,Y 185.251,Z 433.72,A -85,B 0,C 180,E1 -22145.443,E2 -22145.443} C_VEL
LIN {X 0,Y 185.74,Z 424.308,A -85,B 0,C 180,E1 -22148.705,E2 -22148.705} C_VEL
LIN {X 0,Y 186.431,Z 413.012,A -85,B 0,C 180,E1 -22151.965,E2 -22151.965} C_VEL
LIN {X 0,Y 187.36,Z 400.42,A -85,B 0,C 180,E1 -22154.945,E2 -22154.945} C_VEL
LIN {X 0,Y 188.499,Z 386.56,A -85,B 0,C 180,E1 -22157.634,E2 -22157.634} C_VEL
LIN {X 0,Y 189.637,Z 372.918,A -85,B 0,C 180,E1 -22159.766,E2 -22159.766} C_VEL
LIN {X 0,Y 190.686,Z 358.005,A -85,B 0,C 180,E1 -22161.627,E2 -22161.627} C_VEL
LIN {X 0,Y 191.687,Z 341.323,A -85,B 0,C 180,E1 -22163.193,E2 -22163.193} C_VEL
LIN {X 0,Y 192.445,Z 325.03,A -85,B 0,C 180,E1 -22164.33,E2 -22164.33} C_VEL
LIN {X 0,Y 192.68,Z 326.855,A -85,B 0,C 180,E1 -22164.657,E2 -22164.657} C_VEL
LIN {X 0,Y 193.442,Z 326.531,A -85,B 0,C 180,E1 -22165.127,E2 -22165.127} C_VEL
LIN {X 0,Y 194.784,Z 323.7,A -85,B 0,C 180,E1 -22165.735,E2 -22165.735} C_VEL
LIN {X 0,Y 197.232,Z 316.075,A -85,B 0,C 180,E1 -22166.592,E2 -22166.592} C_VEL
LIN {X 0,Y 200.925,Z 302.108,A -85,B 0,C 180,E1 -22167.611,E2 -22167.611} C_VEL
LIN {X 0,Y 203.355,Z 291.838,A -85,B 0,C 180,E1 -22168.162,E2 -22168.162} C_VEL
LIN {X 0,Y 204.911,Z 289.843,A -85,B 0,C 180,E1 -22168.837,E2 -22168.837} C_VEL
LIN {X 0,Y 206.838,Z 285.638,A -85,B 0,C 180,E1 -22169.517,E2 -22169.517} C_VEL
LIN {X 0,Y 209.998,Z 276.263,A -85,B 0,C 180,E1 -22170.411,E2 -22170.411} C_VEL
LIN {X 0,Y 214.082,Z 261.339,A -85,B 0,C 180,E1 -22171.314,E2 -22171.314} C_VEL
LIN {X 0,Y 216.145,Z 253.341,A -85,B 0,C 180,E1 -22171.719,E2 -22171.719} C_VEL
LIN {X 0,Y 219.092,Z 248.97,A -85,B 0,C 180,E1 -22172.705,E2 -22172.705} C_VEL
LIN {X 0,Y 221.883,Z 242.557,A -85,B 0,C 180,E1 -22173.459,E2 -22173.459} C_VEL
LIN {X 0,Y 223.957,Z 236.684,A -85,B 0,C 180,E1 -22173.934,E2 -22173.934} C_VEL
LIN {X 0,Y 224.487,Z 235.949,A -85,B 0,C 180,E1 -22174.097,E2 -22174.097} C_VEL
LIN {X 0,Y 227.98,Z 235.626,A -85,B 0,C 180,E1 -22175.379,E2 -22175.379} C_VEL
LIN {X 0,Y 234.051,Z 246.24,A -85,B 0,C 180,E1 -22177.985,E2 -22177.985} C_VEL
LIN {X 0,Y 239.256,Z 256.382,A -85,B 0,C 180,E1 -22180.052,E2 -22180.052} C_VEL
LIN {X 0,Y 240.336,Z 258.633,A -85,B 0,C 180,E1 -22180.466,E2 -22180.466} C_VEL
LIN {X 0,Y 233.992,Z 353.949,A -85,B 0,C 180,E1 -22183.092,E2 -22183.092} C_VEL
LIN {X 0,Y 232.21,Z 369.32,A -85,B 0,C 180,E1 -22183.824,E2 -22183.824} C_VEL
LIN {X 0,Y 229.953,Z 383.127,A -85,B 0,C 180,E1 -22184.783,E2 -22184.783} C_VEL
LIN {X 0,Y 226.932,Z 397.591,A -85,B 0,C 180,E1 -22186.134,E2 -22186.134} C_VEL
LIN {X 0,Y 223.711,Z 409.517,A -85,B 0,C 180,E1 -22187.509,E2 -22187.509} C_VEL
LIN {X 0,Y 219.701,Z 422.152,A -85,B 0,C 180,E1 -22189.322,E2 -22189.322} C_VEL
LIN {X 0,Y 215.249,Z 433.84,A -85,B 0,C 180,E1 -22191.356,E2 -22191.356} C_VEL
LIN {X 0,Y 210.85,Z 444.633,A -85,B 0,C 180,E1 -22193.724,E2 -22193.724} C_VEL
LIN {X 0,Y 206.505,Z 454.537,A -85,B 0,C 180,E1 -22196.422,E2 -22196.422} C_VEL
LIN {X 0,Y 201.6,Z 464.222,A -85,B 0,C 180,E1 -22199.634,E2 -22199.634} C_VEL
LIN {X 0,Y 196.956,Z 472.995,A -85,B 0,C 180,E1 -22203.355,E2 -22203.355} C_VEL
LIN {X 0,Y 193.763,Z 478.838,A -85,B 0,C 180,E1 -22206.483,E2 -22206.483} C_VEL
LIN {X 0,Y 190.362,Z 484.941,A -85,B 0,C 180,E1 -22210.591,E2 -22210.591} C_VEL
LIN {X 0,Y 187.783,Z 489.643,A -85,B 0,C 180,E1 -22214.81,E2 -22214.81} C_VEL
LIN {X 0,Y 185.821,Z 493.354,A -85,B 0,C 180,E1 -22219.532,E2 -22219.532} C_VEL
LIN {X 0,Y 184.788,Z 495.34,A -85,B 0,C 180,E1 -22223.446,E2 -22223.446} C_VEL
LIN {X 0,Y 184.373,Z 496.472,A -85,B 0,C 180,E1 -22227.813,E2 -22227.813} C_VEL
LIN {X 0,Y 184.371,Z 496.482,A -85,B 0,C 180,E1 -22232.182,E2 -22232.182} C_VEL
LIN {X 0,Y 184.775,Z 495.393,A -85,B 0,C 180,E1 -22236.549,E2 -22236.549} C_VEL
LIN {X 0,Y 185.984,Z 493.174,A -85,B 0,C 180,E1 -22240.888,E2 -22240.888} C_VEL
LIN {X 0,Y 187.762,Z 489.794,A -85,B 0,C 180,E1 -22245.187,E2 -22245.187} C_VEL
LIN {X 0,Y 190.294,Z 485.146,A -85,B 0,C 180,E1 -22249.411,E2 -22249.411} C_VEL
LIN {X 0,Y 193.687,Z 479.09,A -85,B 0,C 180,E1 -22253.521,E2 -22253.521} C_VEL
LIN {X 0,Y 197.836,Z 471.458,A -85,B 0,C 180,E1 -22257.501,E2 -22257.501} C_VEL
LIN {X 0,Y 202.18,Z 463.288,A -85,B 0,C 180,E1 -22260.842,E2 -22260.842} C_VEL
LIN {X 0,Y 206.39,Z 454.974,A -85,B 0,C 180,E1 -22263.593,E2 -22263.593} C_VEL
LIN {X 0,Y 210.732,Z 445.132,A -85,B 0,C 180,E1 -22266.294,E2 -22266.294} C_VEL
LIN {X 0,Y 215.189,Z 434.435,A -85,B 0,C 180,E1 -22268.651,E2 -22268.651} C_VEL
LIN {X 0,Y 219.568,Z 422.873,A -85,B 0,C 180,E1 -22270.702,E2 -22270.702} C_VEL
LIN {X 0,Y 223.575,Z 410.382,A -85,B 0,C 180,E1 -22272.516,E2 -22272.516} C_VEL
LIN {X 0,Y 227.291,Z 396.747,A -85,B 0,C 180,E1 -22274.081,E2 -22274.081} C_VEL
LIN {X 0,Y 230.317,Z 382.078,A -85,B 0,C 180,E1 -22275.426,E2 -22275.426} C_VEL
LIN {X 0,Y 232.647,Z 367.549,A -85,B 0,C 180,E1 -22276.393,E2 -22276.393} C_VEL
LIN {X 0,Y 234.278,Z 352.88,A -85,B 0,C 180,E1 -22277.063,E2 -22277.063} C_VEL
LIN {X 0,Y 239.444,Z 275.599,A -85,B 0,C 180,E1 -22279.186,E2 -22279.186} C_VEL
LIN {X 0,Y 240.538,Z 258.973,A -85,B 0,C 180,E1 -22279.634,E2 -22279.634} C_VEL
LIN {X 0,Y 235.404,Z 248.635,A -85,B 0,C 180,E1 -22281.652,E2 -22281.652} C_VEL
LIN {X 0,Y 229.546,Z 238.184,A -85,B 0,C 180,E1 -22284.122,E2 -22284.122} C_VEL
LIN {X 0,Y 223.792,Z 228.891,A -85,B 0,C 180,E1 -22286.784,E2 -22286.784} C_VEL
LIN {X 0,Y 218.994,Z 221.799,A -85,B 0,C 180,E1 -22289.238,E2 -22289.238} C_VEL
LIN {X 0,Y 214.569,Z 215.588,A -85,B 0,C 180,E1 -22291.758,E2 -22291.758} C_VEL
LIN {X 0,Y 210.451,Z 210.32,A -85,B 0,C 180,E1 -22294.377,E2 -22294.377} C_VEL
LIN {X 0,Y 206.544,Z 205.398,A -85,B 0,C 180,E1 -22297.228,E2 -22297.228} C_VEL
LIN {X 0,Y 203.558,Z 201.807,A -85,B 0,C 180,E1 -22299.736,E2 -22299.736} C_VEL
LIN {X 0,Y 198.468,Z 196.059,A -85,B 0,C 180,E1 -22305.124,E2 -22305.124} C_VEL
LIN {X 0,Y 194.613,Z 191.922,A -85,B 0,C 180,E1 -22311.694,E2 -22311.694} C_VEL
LIN {X 0,Y 194.282,Z 190.218,A -85,B 0,C 180,E1 -22315.851,E2 -22315.851} C_VEL
LIN {X 0,Y 194.322,Z 189.857,A -85,B 0,C 180,E1 -22320,E2 -22320} C_VEL
LIN {X 0,Y 194.512,Z 190.153,A -85,B 0,C 180,E1 -22322.07,E2 -22322.07} C_VEL
LIN {X 0,Y 196.59,Z 194.371,A -85,B 0,C 180,E1 -22330.297,E2 -22330.297} C_VEL
LIN {X 0,Y 197.647,Z 195.636,A -85,B 0,C 180,E1 -22332.319,E2 -22332.319} C_VEL
LIN {X 0,Y 200.744,Z 200.003,A -85,B 0,C 180,E1 -22336.807,E2 -22336.807} C_VEL
LIN {X 0,Y 202.893,Z 202.711,A -85,B 0,C 180,E1 -22338.95,E2 -22338.95} C_VEL
LIN {X 0,Y 206.621,Z 207.19,A -85,B 0,C 180,E1 -22342.101,E2 -22342.101} C_VEL
LIN {X 0,Y 210.105,Z 211.719,A -85,B 0,C 180,E1 -22344.65,E2 -22344.65} C_VEL
LIN {X 0,Y 211.203,Z 214.086,A -85,B 0,C 180,E1 -22345.459,E2 -22345.459} C_VEL
LIN {X 0,Y 212.48,Z 219.285,A -85,B 0,C 180,E1 -22346.541,E2 -22346.541} C_VEL
LIN {X 0,Y 214.064,Z 225.686,A -85,B 0,C 180,E1 -22347.81,E2 -22347.81} C_VEL
LIN {X 0,Y 214.849,Z 227.42,A -85,B 0,C 180,E1 -22348.315,E2 -22348.315} C_VEL
LIN {X 0,Y 221.12,Z 236.941,A -85,B 0,C 180,E1 -22351.722,E2 -22351.722} C_VEL
LIN {X 0,Y 224.228,Z 242.237,A -85,B 0,C 180,E1 -22353.264,E2 -22353.264} C_VEL
LIN {X 0,Y 229.914,Z 258.98,A -85,B 0,C 180,E1 -22356.198,E2 -22356.198} C_VEL
LIN {X 0,Y 232.356,Z 266.519,A -85,B 0,C 180,E1 -22357.374,E2 -22357.374} C_VEL
LIN {X 0,Y 233.286,Z 293.811,A -85,B 0,C 180,E1 -22358.979,E2 -22358.979} C_VEL
LIN {X 0,Y 227.311,Z 379.838,A -85,B 0,C 180,E1 -22361.351,E2 -22361.351} C_VEL
LIN {X 0,Y 225.185,Z 395.243,A -85,B 0,C 180,E1 -22362,E2 -22362} C_VEL
LIN {X 0,Y 222.059,Z 410.754,A -85,B 0,C 180,E1 -22362.959,E2 -22362.959} C_VEL
LIN {X 0,Y 218.122,Z 425.515,A -85,B 0,C 180,E1 -22364.204,E2 -22364.204} C_VEL
LIN {X 0,Y 213.809,Z 438.88,A -85,B 0,C 180,E1 -22365.697,E2 -22365.697} C_VEL
LIN {X 0,Y 209.169,Z 451.242,A -85,B 0,C 180,E1 -22367.457,E2 -22367.457} C_VEL
LIN {X 0,Y 204.434,Z 462.773,A -85,B 0,C 180,E1 -22369.546,E2 -22369.546} C_VEL
LIN {X 0,Y 199.47,Z 473.507,A -85,B 0,C 180,E1 -22371.937,E2 -22371.937} C_VEL
LIN {X 0,Y 194.623,Z 483.469,A -85,B 0,C 180,E1 -22374.71,E2 -22374.71} C_VEL
LIN {X 0,Y 189.666,Z 493.24,A -85,B 0,C 180,E1 -22378.131,E2 -22378.131} C_VEL
LIN {X 0,Y 186.054,Z 500.346,A -85,B 0,C 180,E1 -22381.212,E2 -22381.212} C_VEL
LIN {X 0,Y 182.497,Z 507.285,A -85,B 0,C 180,E1 -22384.941,E2 -22384.941} C_VEL
LIN {X 0,Y 179.452,Z 513.756,A -85,B 0,C 180,E1 -22389.365,E2 -22389.365} C_VEL
LIN {X 0,Y 177.485,Z 518.795,A -85,B 0,C 180,E1 -22393.911,E2 -22393.911} C_VEL
LIN {X 0,Y 176.498,Z 522.521,A -85,B 0,C 180,E1 -22398.519,E2 -22398.519} C_VEL
LIN {X 0,Y 176.528,Z 525.029,A -85,B 0,C 180,E1 -22403.143,E2 -22403.143} C_VEL
LIN {X 0,Y 176.745,Z 525.829,A -85,B 0,C 180,E1 -22405.442,E2 -22405.442} C_VEL
LIN {X 0,Y 177.236,Z 526.504,A -85,B 0,C 180,E1 -22410.003,E2 -22410.003} C_VEL
LIN {X 0,Y 176.773,Z 525.819,A -85,B 0,C 180,E1 -22414.564,E2 -22414.564} C_VEL
LIN {X 0,Y 176.62,Z 525.016,A -85,B 0,C 180,E1 -22416.859,E2 -22416.859} C_VEL
LIN {X 0,Y 176.541,Z 522.484,A -85,B 0,C 180,E1 -22421.484,E2 -22421.484} C_VEL
LIN {X 0,Y 177.494,Z 518.728,A -85,B 0,C 180,E1 -22426.094,E2 -22426.094} C_VEL
LIN {X 0,Y 179.458,Z 513.664,A -85,B 0,C 180,E1 -22430.641,E2 -22430.641} C_VEL
LIN {X 0,Y 182.516,Z 507.176,A -85,B 0,C 180,E1 -22435.063,E2 -22435.063} C_VEL
LIN {X 0,Y 186.65,Z 499.076,A -85,B 0,C 180,E1 -22439.31,E2 -22439.31} C_VEL
LIN {X 0,Y 189.697,Z 493.124,A -85,B 0,C 180,E1 -22441.869,E2 -22441.869} C_VEL
LIN {X 0,Y 196.726,Z 488.77,A -85,B 0,C 180,E1 -22446.122,E2 -22446.122} C_VEL
LIN {X 0,Y 206.153,Z 482.632,A -85,B 0,C 180,E1 -22450.374,E2 -22450.374} C_VEL
LIN {X 0,Y 212.665,Z 478.202,A -85,B 0,C 180,E1 -22452.649,E2 -22452.649} C_VEL
LIN {X 0,Y 222.205,Z 471.463,A -85,B 0,C 180,E1 -22455.371,E2 -22455.371} C_VEL
LIN {X 0,Y 232.489,Z 463.585,A -85,B 0,C 180,E1 -22457.787,E2 -22457.787} C_VEL
LIN {X 0,Y 243.537,Z 454.426,A -85,B 0,C 180,E1 -22459.886,E2 -22459.886} C_VEL
LIN {X 0,Y 244.926,Z 453.231,A -85,B 0,C 180,E1 -22460.111,E2 -22460.111} C_VEL
LIN {X 0,Y 244.244,Z 453.378,A -85,B 0,C 180,E1 -22460.726,E2 -22460.726} C_VEL
LIN {X 0,Y 236.667,Z 458.041,A -85,B 0,C 180,E1 -22462.5,E2 -22462.5} C_VEL
LIN {X 0,Y 227.122,Z 463.01,A -85,B 0,C 180,E1 -22465.078,E2 -22465.078} C_VEL
LIN {X 0,Y 220.372,Z 465.836,A -85,B 0,C 180,E1 -22467.17,E2 -22467.17} C_VEL
LIN {X 0,Y 211.966,Z 468.52,A -85,B 0,C 180,E1 -22470.176,E2 -22470.176} C_VEL
LIN {X 0,Y 204.381,Z 469.913,A -85,B 0,C 180,E1 -22473.447,E2 -22473.447} C_VEL
LIN {X 0,Y 197.611,Z 470.051,A -85,B 0,C 180,E1 -22476.97,E2 -22476.97} C_VEL
LIN {X 0,Y 191.719,Z 468.863,A -85,B 0,C 180,E1 -22480.736,E2 -22480.736} C_VEL
LIN {X 0,Y 186.9,Z 466.287,A -85,B 0,C 180,E1 -22484.739,E2 -22484.739} C_VEL
LIN {X 0,Y 183.279,Z 462.297,A -85,B 0,C 180,E1 -22488.947,E2 -22488.947} C_VEL
LIN {X 0,Y 181.275,Z 458.357,A -85,B 0,C 180,E1 -22492.201,E2 -22492.201} C_VEL
LIN {X 0,Y 179.321,Z 451.649,A -85,B 0,C 180,E1 -22496.63,E2 -22496.63} C_VEL
LIN {X 0,Y 178.427,Z 444.28,A -85,B 0,C 180,E1 -22500.564,E2 -22500.564} C_VEL
LIN {X 0,Y 178.227,Z 435.314,A -85,B 0,C 180,E1 -22504.524,E2 -22504.524} C_VEL
LIN {X 0,Y 178.56,Z 426.011,A -85,B 0,C 180,E1 -22507.918,E2 -22507.918} C_VEL
LIN {X 0,Y 179.265,Z 413.869,A -85,B 0,C 180,E1 -22511.591,E2 -22511.591} C_VEL
LIN {X 0,Y 180.191,Z 401.296,A -85,B 0,C 180,E1 -22514.686,E2 -22514.686} C_VEL
LIN {X 0,Y 181.306,Z 387.501,A -85,B 0,C 180,E1 -22517.483,E2 -22517.483} C_VEL
LIN {X 0,Y 182.459,Z 373.895,A -85,B 0,C 180,E1 -22519.697,E2 -22519.697} C_VEL
LIN {X 0,Y 183.308,Z 361.859,A -85,B 0,C 180,E1 -22521.36,E2 -22521.36} C_VEL
LIN {X 0,Y 183.465,Z 362.922,A -85,B 0,C 180,E1 -22521.636,E2 -22521.636} C_VEL
LIN {X 0,Y 183.922,Z 363.044,A -85,B 0,C 180,E1 -22522.022,E2 -22522.022} C_VEL
LIN {X 0,Y 185.05,Z 361.499,A -85,B 0,C 180,E1 -22522.698,E2 -22522.698} C_VEL
LIN {X 0,Y 187.153,Z 356.884,A -85,B 0,C 180,E1 -22523.678,E2 -22523.678} C_VEL
LIN {X 0,Y 189.328,Z 350.429,A -85,B 0,C 180,E1 -22524.538,E2 -22524.538} C_VEL
LIN {X 0,Y 192.271,Z 339.554,A -85,B 0,C 180,E1 -22525.508,E2 -22525.508} C_VEL
LIN {X 0,Y 193.822,Z 333.16,A -85,B 0,C 180,E1 -22525.937,E2 -22525.937} C_VEL
LIN {X 0,Y 195.405,Z 330.938,A -85,B 0,C 180,E1 -22526.716,E2 -22526.716} C_VEL
LIN {X 0,Y 197.089,Z 327.226,A -85,B 0,C 180,E1 -22527.402,E2 -22527.402} C_VEL
LIN {X 0,Y 199.754,Z 319.27,A -85,B 0,C 180,E1 -22528.275,E2 -22528.275} C_VEL
LIN {X 0,Y 203.36,Z 306.221,A -85,B 0,C 180,E1 -22529.219,E2 -22529.219} C_VEL
LIN {X 0,Y 205.929,Z 296.157,A -85,B 0,C 180,E1 -22529.802,E2 -22529.802} C_VEL
LIN {X 0,Y 208.201,Z 292.196,A -85,B 0,C 180,E1 -22530.631,E2 -22530.631} C_VEL
LIN {X 0,Y 210.929,Z 285.38,A -85,B 0,C 180,E1 -22531.444,E2 -22531.444} C_VEL
LIN {X 0,Y 214.693,Z 273.424,A -85,B 0,C 180,E1 -22532.345,E2 -22532.345} C_VEL
LIN {X 0,Y 219.046,Z 257.416,A -85,B 0,C 180,E1 -22533.192,E2 -22533.192} C_VEL
LIN {X 0,Y 222.1,Z 252.52,A -85,B 0,C 180,E1 -22534.12,E2 -22534.12} C_VEL
LIN {X 0,Y 225.263,Z 245.256,A -85,B 0,C 180,E1 -22534.912,E2 -22534.912} C_VEL
LIN {X 0,Y 226.095,Z 243.177,A -85,B 0,C 180,E1 -22535.104,E2 -22535.104} C_VEL
LIN {X 0,Y 231.432,Z 252.922,A -85,B 0,C 180,E1 -22537.471,E2 -22537.471} C_VEL
LIN {X 0,Y 235.672,Z 261.541,A -85,B 0,C 180,E1 -22539.232,E2 -22539.232} C_VEL
LIN {X 0,Y 229.212,Z 354.474,A -85,B 0,C 180,E1 -22541.799,E2 -22541.799} C_VEL
LIN {X 0,Y 227.371,Z 369.94,A -85,B 0,C 180,E1 -22542.545,E2 -22542.545} C_VEL
LIN {X 0,Y 224.859,Z 384.731,A -85,B 0,C 180,E1 -22543.595,E2 -22543.595} C_VEL
LIN {X 0,Y 221.892,Z 398.161,A -85,B 0,C 180,E1 -22544.869,E2 -22544.869} C_VEL
LIN {X 0,Y 218.554,Z 410.091,A -85,B 0,C 180,E1 -22546.258,E2 -22546.258} C_VEL
LIN {X 0,Y 214.382,Z 422.73,A -85,B 0,C 180,E1 -22548.089,E2 -22548.089} C_VEL
LIN {X 0,Y 209.767,Z 434.42,A -85,B 0,C 180,E1 -22550.149,E2 -22550.149} C_VEL
LIN {X 0,Y 205.173,Z 445.216,A -85,B 0,C 180,E1 -22552.552,E2 -22552.552} C_VEL
LIN {X 0,Y 200.654,Z 455.119,A -85,B 0,C 180,E1 -22555.305,E2 -22555.305} C_VEL
LIN {X 0,Y 195.526,Z 464.805,A -85,B 0,C 180,E1 -22558.585,E2 -22558.585} C_VEL
LIN {X 0,Y 191.176,Z 472.588,A -85,B 0,C 180,E1 -22561.92,E2 -22561.92} C_VEL
LIN {X 0,Y 187.297,Z 479.423,A -85,B 0,C 180,E1 -22565.619,E2 -22565.619} C_VEL
LIN {X 0,Y 183.682,Z 485.527,A -85,B 0,C 180,E1 -22569.855,E2 -22569.855} C_VEL
LIN {X 0,Y 180.96,Z 490.229,A -85,B 0,C 180,E1 -22574.222,E2 -22574.222} C_VEL
LIN {X 0,Y 178.811,Z 494.049,A -85,B 0,C 180,E1 -22579.298,E2 -22579.298} C_VEL
LIN {X 0,Y 177.761,Z 495.925,A -85,B 0,C 180,E1 -22583.185,E2 -22583.185} C_VEL
LIN {X 0,Y 177.3,Z 497.057,A -85,B 0,C 180,E1 -22587.725,E2 -22587.725} C_VEL
LIN {X 0,Y 177.298,Z 497.067,A -85,B 0,C 180,E1 -22592.269,E2 -22592.269} C_VEL
LIN {X 0,Y 177.749,Z 495.977,A -85,B 0,C 180,E1 -22596.809,E2 -22596.809} C_VEL
LIN {X 0,Y 179.023,Z 493.759,A -85,B 0,C 180,E1 -22601.317,E2 -22601.317} C_VEL
LIN {X 0,Y 180.935,Z 490.378,A -85,B 0,C 180,E1 -22605.774,E2 -22605.774} C_VEL
LIN {X 0,Y 183.621,Z 485.73,A -85,B 0,C 180,E1 -22610.146,E2 -22610.146} C_VEL
LIN {X 0,Y 187.216,Z 479.672,A -85,B 0,C 180,E1 -22614.386,E2 -22614.386} C_VEL
LIN {X 0,Y 191.588,Z 472.038,A -85,B 0,C 180,E1 -22618.478,E2 -22618.478} C_VEL
LIN {X 0,Y 196.133,Z 463.868,A -85,B 0,C 180,E1 -22621.903,E2 -22621.903} C_VEL
LIN {X 0,Y 200.533,Z 455.552,A -85,B 0,C 180,E1 -22624.712,E2 -22624.712} C_VEL
LIN {X 0,Y 205.076,Z 445.707,A -85,B 0,C 180,E1 -22627.463,E2 -22627.463} C_VEL
LIN {X 0,Y 209.702,Z 435.009,A -85,B 0,C 180,E1 -22629.86,E2 -22629.86} C_VEL
LIN {X 0,Y 214.267,Z 423.441,A -85,B 0,C 180,E1 -22631.933,E2 -22631.933} C_VEL
LIN {X 0,Y 218.428,Z 410.945,A -85,B 0,C 180,E1 -22633.767,E2 -22633.767} C_VEL
LIN {X 0,Y 222.265,Z 397.305,A -85,B 0,C 180,E1 -22635.349,E2 -22635.349} C_VEL
LIN {X 0,Y 225.36,Z 382.937,A -85,B 0,C 180,E1 -22636.679,E2 -22636.679} C_VEL
LIN {X 0,Y 227.821,Z 368.096,A -85,B 0,C 180,E1 -22637.681,E2 -22637.681} C_VEL
LIN {X 0,Y 229.518,Z 353.368,A -85,B 0,C 180,E1 -22638.356,E2 -22638.356} C_VEL
LIN {X 0,Y 233.897,Z 290.452,A -85,B 0,C 180,E1 -22640.103,E2 -22640.103} C_VEL
LIN {X 0,Y 235.797,Z 261.605,A -85,B 0,C 180,E1 -22640.905,E2 -22640.905} C_VEL
LIN {X 0,Y 230.422,Z 250.779,A -85,B 0,C 180,E1 -22643.163,E2 -22643.163} C_VEL
LIN {X 0,Y 223.677,Z 238.933,A -85,B 0,C 180,E1 -22646.25,E2 -22646.25} C_VEL
LIN {X 0,Y 217.404,Z 228.998,A -85,B 0,C 180,E1 -22649.493,E2 -22649.493} C_VEL
LIN {X 0,Y 211.567,Z 220.758,A -85,B 0,C 180,E1 -22652.955,E2 -22652.955} C_VEL
LIN {X 0,Y 208.259,Z 216.479,A -85,B 0,C 180,E1 -22655.182,E2 -22655.182} C_VEL
LIN {X 0,Y 204.955,Z 212.111,A -85,B 0,C 180,E1 -22657.707,E2 -22657.707} C_VEL
LIN {X 0,Y 201.941,Z 208.384,A -85,B 0,C 180,E1 -22660.341,E2 -22660.341} C_VEL
LIN {X 0,Y 197.225,Z 202.883,A -85,B 0,C 180,E1 -22665.555,E2 -22665.555} C_VEL
LIN {X 0,Y 193.03,Z 198.198,A -85,B 0,C 180,E1 -22673.467,E2 -22673.467} C_VEL
LIN {X 0,Y 192.31,Z 196.921,A -85,B 0,C 180,E1 -22676.857,E2 -22676.857} C_VEL
LIN {X 0,Y 192.18,Z 196.759,A -85,B 0,C 180,E1 -22681.047,E2 -22681.047} C_VEL
LIN {X 0,Y 192.598,Z 197.94,A -85,B 0,C 180,E1 -22684.185,E2 -22684.185} C_VEL
LIN {X 0,Y 196.201,Z 202.708,A -85,B 0,C 180,E1 -22692.279,E2 -22692.279} C_VEL
LIN {X 0,Y 200.72,Z 208.391,A -85,B 0,C 180,E1 -22697.751,E2 -22697.751} C_VEL
LIN {X 0,Y 204.883,Z 213.71,A -85,B 0,C 180,E1 -22701.506,E2 -22701.506} C_VEL
LIN {X 0,Y 209.473,Z 219.918,A -85,B 0,C 180,E1 -22704.928,E2 -22704.928} C_VEL
LIN {X 0,Y 214.849,Z 227.42,A -85,B 0,C 180,E1 -22708.315,E2 -22708.315} C_VEL
LIN {X 0,Y 216.64,Z 231.262,A -85,B 0,C 180,E1 -22709.418,E2 -22709.418} C_VEL
LIN {X 0,Y 219.028,Z 238.899,A -85,B 0,C 180,E1 -22710.962,E2 -22710.962} C_VEL
LIN {X 0,Y 222.526,Z 252.115,A -85,B 0,C 180,E1 -22713.169,E2 -22713.169} C_VEL
LIN {X 0,Y 226.676,Z 265.093,A -85,B 0,C 180,E1 -22715.408,E2 -22715.408} C_VEL
LIN {X 0,Y 228.061,Z 269.468,A -85,B 0,C 180,E1 -22716.114,E2 -22716.114} C_VEL
LIN {X 0,Y 228.771,Z 294.637,A -85,B 0,C 180,E1 -22717.624,E2 -22717.624} C_VEL
LIN {X 0,Y 222.676,Z 379.349,A -85,B 0,C 180,E1 -22719.977,E2 -22719.977} C_VEL
LIN {X 0,Y 220.493,Z 394.712,A -85,B 0,C 180,E1 -22720.628,E2 -22720.628} C_VEL
LIN {X 0,Y 217.282,Z 410.204,A -85,B 0,C 180,E1 -22721.588,E2 -22721.588} C_VEL
LIN {X 0,Y 213.21,Z 424.952,A -85,B 0,C 180,E1 -22722.83,E2 -22722.83} C_VEL
LIN {X 0,Y 208.784,Z 438.312,A -85,B 0,C 180,E1 -22724.336,E2 -22724.336} C_VEL
LIN {X 0,Y 203.964,Z 450.667,A -85,B 0,C 180,E1 -22726.1,E2 -22726.1} C_VEL
LIN {X 0,Y 198.563,Z 463.263,A -85,B 0,C 180,E1 -22728.426,E2 -22728.426} C_VEL
LIN {X 0,Y 192.987,Z 474.714,A -85,B 0,C 180,E1 -22731.087,E2 -22731.087} C_VEL
LIN {X 0,Y 188.019,Z 484.383,A -85,B 0,C 180,E1 -22733.937,E2 -22733.937} C_VEL
LIN {X 0,Y 182.904,Z 493.898,A -85,B 0,C 180,E1 -22737.46,E2 -22737.46} C_VEL
LIN {X 0,Y 178.627,Z 501.844,A -85,B 0,C 180,E1 -22741.189,E2 -22741.189} C_VEL
LIN {X 0,Y 175.067,Z 508.457,A -85,B 0,C 180,E1 -22745.073,E2 -22745.073} C_VEL
LIN {X 0,Y 172.734,Z 513.163,A -85,B 0,C 180,E1 -22748.523,E2 -22748.523} C_VEL
LIN {X 0,Y 170.572,Z 518.201,A -85,B 0,C 180,E1 -22753.24,E2 -22753.24} C_VEL
LIN {X 0,Y 169.469,Z 521.929,A -85,B 0,C 180,E1 -22758.036,E2 -22758.036} C_VEL
LIN {X 0,Y 169.416,Z 524.437,A -85,B 0,C 180,E1 -22762.854,E2 -22762.854} C_VEL
LIN {X 0,Y 169.649,Z 525.24,A -85,B 0,C 180,E1 -22765.25,E2 -22765.25} C_VEL
LIN {X 0,Y 170.144,Z 525.918,A -85,B 0,C 180,E1 -22770.003,E2 -22770.003} C_VEL
LIN {X 0,Y 169.681,Z 525.231,A -85,B 0,C 180,E1 -22774.755,E2 -22774.755} C_VEL
LIN {X 0,Y 169.505,Z 524.424,A -85,B 0,C 180,E1 -22777.148,E2 -22777.148} C_VEL
LIN {X 0,Y 169.506,Z 521.89,A -85,B 0,C 180,E1 -22781.968,E2 -22781.968} C_VEL
LIN {X 0,Y 170.577,Z 518.132,A -85,B 0,C 180,E1 -22786.766,E2 -22786.766} C_VEL
LIN {X 0,Y 172.743,Z 513.069,A -85,B 0,C 180,E1 -22791.482,E2 -22791.482} C_VEL
LIN {X 0,Y 176.016,Z 506.581,A -85,B 0,C 180,E1 -22796.056,E2 -22796.056} C_VEL
LIN {X 0,Y 180.383,Z 498.479,A -85,B 0,C 180,E1 -22800.434,E2 -22800.434} C_VEL
LIN {X 0,Y 183.823,Z 492.357,A -85,B 0,C 180,E1 -22803.178,E2 -22803.178} C_VEL
LIN {X 0,Y 191.007,Z 488.519,A -85,B 0,C 180,E1 -22807.384,E2 -22807.384} C_VEL
LIN {X 0,Y 200.795,Z 482.898,A -85,B 0,C 180,E1 -22811.686,E2 -22811.686} C_VEL
LIN {X 0,Y 207.525,Z 478.872,A -85,B 0,C 180,E1 -22813.97,E2 -22813.97} C_VEL
LIN {X 0,Y 219.873,Z 470.931,A -85,B 0,C 180,E1 -22817.324,E2 -22817.324} C_VEL
LIN {X 0,Y 232.056,Z 462.337,A -85,B 0,C 180,E1 -22819.884,E2 -22819.884} C_VEL
LIN {X 0,Y 234.718,Z 460.35,A -85,B 0,C 180,E1 -22820.376,E2 -22820.376} C_VEL
LIN {X 0,Y 234.179,Z 460.38,A -85,B 0,C 180,E1 -22820.933,E2 -22820.933} C_VEL
LIN {X 0,Y 224.172,Z 465.089,A -85,B 0,C 180,E1 -22823.44,E2 -22823.44} C_VEL
LIN {X 0,Y 214.797,Z 468.536,A -85,B 0,C 180,E1 -22826.205,E2 -22826.205} C_VEL
LIN {X 0,Y 206.102,Z 470.737,A -85,B 0,C 180,E1 -22829.237,E2 -22829.237} C_VEL
LIN {X 0,Y 198.251,Z 471.67,A -85,B 0,C 180,E1 -22832.558,E2 -22832.558} C_VEL
LIN {X 0,Y 191.208,Z 471.357,A -85,B 0,C 180,E1 -22836.152,E2 -22836.152} C_VEL
LIN {X 0,Y 185.083,Z 469.749,A -85,B 0,C 180,E1 -22840.017,E2 -22840.017} C_VEL
LIN {X 0,Y 180.091,Z 466.792,A -85,B 0,C 180,E1 -22844.147,E2 -22844.147} C_VEL
LIN {X 0,Y 176.345,Z 462.434,A -85,B 0,C 180,E1 -22848.506,E2 -22848.506} C_VEL
LIN {X 0,Y 174.245,Z 458.17,A -85,B 0,C 180,E1 -22851.885,E2 -22851.885} C_VEL
LIN {X 0,Y 172.644,Z 452.99,A -85,B 0,C 180,E1 -22855.33,E2 -22855.33} C_VEL
LIN {X 0,Y 171.403,Z 444.551,A -85,B 0,C 180,E1 -22860,E2 -22860} C_VEL
LIN {X 0,Y 171.2,Z 435.334,A -85,B 0,C 180,E1 -22864.12,E2 -22864.12} C_VEL
LIN {X 0,Y 171.572,Z 424.181,A -85,B 0,C 180,E1 -22868.243,E2 -22868.243} C_VEL
LIN {X 0,Y 172.259,Z 412.475,A -85,B 0,C 180,E1 -22871.771,E2 -22871.771} C_VEL
LIN {X 0,Y 173.207,Z 399.53,A -85,B 0,C 180,E1 -22874.991,E2 -22874.991} C_VEL
LIN {X 0,Y 174.266,Z 386.673,A -85,B 0,C 180,E1 -22877.606,E2 -22877.606} C_VEL
LIN {X 0,Y 174.549,Z 383.653,A -85,B 0,C 180,E1 -22878.183,E2 -22878.183} C_VEL
LIN {X 0,Y 174.64,Z 384.238,A -85,B 0,C 180,E1 -22878.477,E2 -22878.477} C_VEL
LIN {X 0,Y 175.293,Z 384.261,A -85,B 0,C 180,E1 -22879.163,E2 -22879.163} C_VEL
LIN {X 0,Y 176.947,Z 382.309,A -85,B 0,C 180,E1 -22880.185,E2 -22880.185} C_VEL
LIN {X 0,Y 179.58,Z 377.971,A -85,B 0,C 180,E1 -22881.375,E2 -22881.375} C_VEL
LIN {X 0,Y 182.831,Z 371.021,A -85,B 0,C 180,E1 -22882.533,E2 -22882.533} C_VEL
LIN {X 0,Y 183.386,Z 369.737,A -85,B 0,C 180,E1 -22882.741,E2 -22882.741} C_VEL
LIN {X 0,Y 185.109,Z 367.962,A -85,B 0,C 180,E1 -22883.749,E2 -22883.749} C_VEL
LIN {X 0,Y 187.547,Z 363.902,A -85,B 0,C 180,E1 -22884.842,E2 -22884.842} C_VEL
LIN {X 0,Y 190.418,Z 357.166,A -85,B 0,C 180,E1 -22885.921,E2 -22885.921} C_VEL
LIN {X 0,Y 193.518,Z 347.27,A -85,B 0,C 180,E1 -22886.926,E2 -22886.926} C_VEL
LIN {X 0,Y 196.052,Z 337.659,A -85,B 0,C 180,E1 -22887.631,E2 -22887.631} C_VEL
LIN {X 0,Y 198.586,Z 333.092,A -85,B 0,C 180,E1 -22888.684,E2 -22888.684} C_VEL
LIN {X 0,Y 201.055,Z 326.752,A -85,B 0,C 180,E1 -22889.516,E2 -22889.516} C_VEL
LIN {X 0,Y 205.011,Z 313.767,A -85,B 0,C 180,E1 -22890.572,E2 -22890.572} C_VEL
LIN {X 0,Y 208.592,Z 300.132,A -85,B 0,C 180,E1 -22891.342,E2 -22891.342} C_VEL
LIN {X 0,Y 211.324,Z 295.021,A -85,B 0,C 180,E1 -22892.239,E2 -22892.239} C_VEL
LIN {X 0,Y 214.438,Z 287.123,A -85,B 0,C 180,E1 -22893.081,E2 -22893.081} C_VEL
LIN {X 0,Y 218.397,Z 274.632,A -85,B 0,C 180,E1 -22893.947,E2 -22893.947} C_VEL
LIN {X 0,Y 222.084,Z 261.282,A -85,B 0,C 180,E1 -22894.613,E2 -22894.613} C_VEL
LIN {X 0,Y 225.243,Z 256.035,A -85,B 0,C 180,E1 -22895.496,E2 -22895.496} C_VEL
LIN {X 0,Y 225.96,Z 254.55,A -85,B 0,C 180,E1 -22895.675,E2 -22895.675} C_VEL
LIN {X 0,Y 226.226,Z 254.426,A -85,B 0,C 180,E1 -22895.763,E2 -22895.763} C_VEL
LIN {X 0,Y 231.135,Z 264.401,A -85,B 0,C 180,E1 -22897.952,E2 -22897.952} C_VEL
LIN {X 0,Y 224.565,Z 354.998,A -85,B 0,C 180,E1 -22900.455,E2 -22900.455} C_VEL
LIN {X 0,Y 222.642,Z 370.614,A -85,B 0,C 180,E1 -22901.213,E2 -22901.213} C_VEL
LIN {X 0,Y 220,Z 385.568,A -85,B 0,C 180,E1 -22902.287,E2 -22902.287} C_VEL
LIN {X 0,Y 216.965,Z 398.731,A -85,B 0,C 180,E1 -22903.547,E2 -22903.547} C_VEL
LIN {X 0,Y 213.511,Z 410.664,A -85,B 0,C 180,E1 -22904.949,E2 -22904.949} C_VEL
LIN {X 0,Y 209.179,Z 423.306,A -85,B 0,C 180,E1 -22906.796,E2 -22906.796} C_VEL
LIN {X 0,Y 204.4,Z 434.998,A -85,B 0,C 180,E1 -22908.881,E2 -22908.881} C_VEL
LIN {X 0,Y 199.588,Z 445.799,A -85,B 0,C 180,E1 -22911.313,E2 -22911.313} C_VEL
LIN {X 0,Y 194.885,Z 455.701,A -85,B 0,C 180,E1 -22914.123,E2 -22914.123} C_VEL
LIN {X 0,Y 189.524,Z 465.389,A -85,B 0,C 180,E1 -22917.47,E2 -22917.47} C_VEL
LIN {X 0,Y 184.861,Z 473.355,A -85,B 0,C 180,E1 -22920.976,E2 -22920.976} C_VEL
LIN {X 0,Y 180.875,Z 480.007,A -85,B 0,C 180,E1 -22924.694,E2 -22924.694} C_VEL
LIN {X 0,Y 177.042,Z 486.113,A -85,B 0,C 180,E1 -22929.064,E2 -22929.064} C_VEL
LIN {X 0,Y 174.16,Z 490.814,A -85,B 0,C 180,E1 -22933.589,E2 -22933.589} C_VEL
LIN {X 0,Y 172.08,Z 494.25,A -85,B 0,C 180,E1 -22938.214,E2 -22938.214} C_VEL
LIN {X 0,Y 170.741,Z 496.51,A -85,B 0,C 180,E1 -22942.904,E2 -22942.904} C_VEL
LIN {X 0,Y 170.228,Z 497.642,A -85,B 0,C 180,E1 -22947.631,E2 -22947.631} C_VEL
LIN {X 0,Y 170.226,Z 497.652,A -85,B 0,C 180,E1 -22952.363,E2 -22952.363} C_VEL
LIN {X 0,Y 170.73,Z 496.561,A -85,B 0,C 180,E1 -22957.091,E2 -22957.091} C_VEL
LIN {X 0,Y 172.08,Z 494.344,A -85,B 0,C 180,E1 -22961.78,E2 -22961.78} C_VEL
LIN {X 0,Y 174.133,Z 490.962,A -85,B 0,C 180,E1 -22966.407,E2 -22966.407} C_VEL
LIN {X 0,Y 176.985,Z 486.314,A -85,B 0,C 180,E1 -22970.936,E2 -22970.936} C_VEL
LIN {X 0,Y 180.791,Z 480.254,A -85,B 0,C 180,E1 -22975.313,E2 -22975.313} C_VEL
LIN {X 0,Y 185.385,Z 472.62,A -85,B 0,C 180,E1 -22979.523,E2 -22979.523} C_VEL
LIN {X 0,Y 190.152,Z 464.448,A -85,B 0,C 180,E1 -22983.032,E2 -22983.032} C_VEL
LIN {X 0,Y 194.754,Z 456.13,A -85,B 0,C 180,E1 -22985.899,E2 -22985.899} C_VEL
LIN {X 0,Y 199.511,Z 446.282,A -85,B 0,C 180,E1 -22988.698,E2 -22988.698} C_VEL
LIN {X 0,Y 204.336,Z 435.581,A -85,B 0,C 180,E1 -22991.128,E2 -22991.128} C_VEL
LIN {X 0,Y 209.068,Z 424.01,A -85,B 0,C 180,E1 -22993.226,E2 -22993.226} C_VEL
LIN {X 0,Y 213.393,Z 411.508,A -85,B 0,C 180,E1 -22995.076,E2 -22995.076} C_VEL
LIN {X 0,Y 217.355,Z 397.862,A -85,B 0,C 180,E1 -22996.675,E2 -22996.675} C_VEL
LIN {X 0,Y 220.476,Z 383.948,A -85,B 0,C 180,E1 -22997.978,E2 -22997.978} C_VEL
LIN {X 0,Y 223.12,Z 368.635,A -85,B 0,C 180,E1 -22999.023,E2 -22999.023} C_VEL
LIN {X 0,Y 224.875,Z 353.851,A -85,B 0,C 180,E1 -22999.704,E2 -22999.704} C_VEL
LIN {X 0,Y 229.284,Z 292.619,A -85,B 0,C 180,E1 -23001.417,E2 -23001.417} C_VEL
LIN {X 0,Y 231.257,Z 264.559,A -85,B 0,C 180,E1 -23002.186,E2 -23002.186} C_VEL
LIN {X 0,Y 226.163,Z 254.253,A -85,B 0,C 180,E1 -23004.465,E2 -23004.465} C_VEL
LIN {X 0,Y 219.8,Z 242.877,A -85,B 0,C 180,E1 -23007.581,E2 -23007.581} C_VEL
LIN {X 0,Y 214.407,Z 234.271,A -85,B 0,C 180,E1 -23010.549,E2 -23010.549} C_VEL
LIN {X 0,Y 209.087,Z 226.595,A -85,B 0,C 180,E1 -23013.888,E2 -23013.888} C_VEL
LIN {X 0,Y 206.452,Z 223.007,A -85,B 0,C 180,E1 -23015.755,E2 -23015.755} C_VEL
LIN {X 0,Y 203.096,Z 218.546,A -85,B 0,C 180,E1 -23018.428,E2 -23018.428} C_VEL
LIN {X 0,Y 199.542,Z 214.134,A -85,B 0,C 180,E1 -23021.752,E2 -23021.752} C_VEL
LIN {X 0,Y 195.777,Z 209.464,A -85,B 0,C 180,E1 -23026.296,E2 -23026.296} C_VEL
LIN {X 0,Y 192.085,Z 205.191,A -85,B 0,C 180,E1 -23033.698,E2 -23033.698} C_VEL
LIN {X 0,Y 191.445,Z 203.973,A -85,B 0,C 180,E1 -23036.843,E2 -23036.843} C_VEL
LIN {X 0,Y 191.317,Z 203.79,A -85,B 0,C 180,E1 -23041.052,E2 -23041.052} C_VEL
LIN {X 0,Y 191.763,Z 205.204,A -85,B 0,C 180,E1 -23044.401,E2 -23044.401} C_VEL
LIN {X 0,Y 194.999,Z 209.553,A -85,B 0,C 180,E1 -23051.828,E2 -23051.828} C_VEL
LIN {X 0,Y 199.295,Z 215.148,A -85,B 0,C 180,E1 -23057.262,E2 -23057.262} C_VEL
LIN {X 0,Y 203.201,Z 220.332,A -85,B 0,C 180,E1 -23060.935,E2 -23060.935} C_VEL
LIN {X 0,Y 206.902,Z 225.499,A -85,B 0,C 180,E1 -23063.847,E2 -23063.847} C_VEL
LIN {X 0,Y 209.813,Z 229.738,A -85,B 0,C 180,E1 -23065.875,E2 -23065.875} C_VEL
LIN {X 0,Y 213.015,Z 234.336,A -85,B 0,C 180,E1 -23067.887,E2 -23067.887} C_VEL
LIN {X 0,Y 218.388,Z 242.733,A -85,B 0,C 180,E1 -23070.923,E2 -23070.923} C_VEL
LIN {X 0,Y 220.971,Z 247.33,A -85,B 0,C 180,E1 -23072.277,E2 -23072.277} C_VEL
LIN {X 0,Y 222.526,Z 252.115,A -85,B 0,C 180,E1 -23073.169,E2 -23073.169} C_VEL
LIN {X 0,Y 223.668,Z 257.222,A -85,B 0,C 180,E1 -23073.892,E2 -23073.892} C_VEL
LIN {X 0,Y 224.221,Z 262.822,A -85,B 0,C 180,E1 -23074.407,E2 -23074.407} C_VEL
LIN {X 0,Y 224.262,Z 274.699,A -85,B 0,C 180,E1 -23075.067,E2 -23075.067} C_VEL
LIN {X 0,Y 224.126,Z 282.729,A -85,B 0,C 180,E1 -23075.45,E2 -23075.45} C_VEL
LIN {X 0,Y 224.35,Z 296.5,A -85,B 0,C 180,E1 -23076.256,E2 -23076.256} C_VEL
LIN {X 0,Y 218.184,Z 378.86,A -85,B 0,C 180,E1 -23078.548,E2 -23078.548} C_VEL
LIN {X 0,Y 215.935,Z 394.181,A -85,B 0,C 180,E1 -23079.198,E2 -23079.198} C_VEL
LIN {X 0,Y 212.629,Z 409.654,A -85,B 0,C 180,E1 -23080.155,E2 -23080.155} C_VEL
LIN {X 0,Y 208.438,Z 424.39,A -85,B 0,C 180,E1 -23081.395,E2 -23081.395} C_VEL
LIN {X 0,Y 203.858,Z 437.741,A -85,B 0,C 180,E1 -23082.9,E2 -23082.9} C_VEL
LIN {X 0,Y 198.874,Z 450.09,A -85,B 0,C 180,E1 -23084.672,E2 -23084.672} C_VEL
LIN {X 0,Y 193.291,Z 462.685,A -85,B 0,C 180,E1 -23087.024,E2 -23087.024} C_VEL
LIN {X 0,Y 187.47,Z 474.13,A -85,B 0,C 180,E1 -23089.712,E2 -23089.712} C_VEL
LIN {X 0,Y 182.264,Z 483.796,A -85,B 0,C 180,E1 -23092.609,E2 -23092.609} C_VEL
LIN {X 0,Y 176.888,Z 493.309,A -85,B 0,C 180,E1 -23096.208,E2 -23096.208} C_VEL
LIN {X 0,Y 172.946,Z 500.224,A -85,B 0,C 180,E1 -23099.476,E2 -23099.476} C_VEL
LIN {X 0,Y 168.569,Z 507.865,A -85,B 0,C 180,E1 -23104.042,E2 -23104.042} C_VEL
LIN {X 0,Y 165.286,Z 514.1,A -85,B 0,C 180,E1 -23108.947,E2 -23108.947} C_VEL
LIN {X 0,Y 163.291,Z 518.69,A -85,B 0,C 180,E1 -23113.758,E2 -23113.758} C_VEL
LIN {X 0,Y 162.445,Z 521.335,A -85,B 0,C 180,E1 -23117.51,E2 -23117.51} C_VEL
LIN {X 0,Y 162.294,Z 523.844,A -85,B 0,C 180,E1 -23122.539,E2 -23122.539} C_VEL
LIN {X 0,Y 162.554,Z 524.652,A -85,B 0,C 180,E1 -23125.043,E2 -23125.043} C_VEL
LIN {X 0,Y 163.051,Z 525.332,A -85,B 0,C 180,E1 -23130.003,E2 -23130.003} C_VEL
LIN {X 0,Y 162.592,Z 524.642,A -85,B 0,C 180,E1 -23134.962,E2 -23134.962} C_VEL
LIN {X 0,Y 162.287,Z 522.712,A -85,B 0,C 180,E1 -23139.978,E2 -23139.978} C_VEL
LIN {X 0,Y 162.966,Z 519.575,A -85,B 0,C 180,E1 -23144.999,E2 -23144.999} C_VEL
LIN {X 0,Y 164.878,Z 514.794,A -85,B 0,C 180,E1 -23150.322,E2 -23150.322} C_VEL
LIN {X 0,Y 167.671,Z 509.418,A -85,B 0,C 180,E1 -23154.784,E2 -23154.784} C_VEL
LIN {X 0,Y 171.796,Z 502.155,A -85,B 0,C 180,E1 -23159.403,E2 -23159.403} C_VEL
LIN {X 0,Y 176.185,Z 494.37,A -85,B 0,C 180,E1 -23163.279,E2 -23163.279} C_VEL
LIN {X 0,Y 178.083,Z 491.551,A -85,B 0,C 180,E1 -23164.566,E2 -23164.566} C_VEL
LIN {X 0,Y 187.302,Z 487.269,A -85,B 0,C 180,E1 -23169.637,E2 -23169.637} C_VEL
LIN {X 0,Y 197.794,Z 481.913,A -85,B 0,C 180,E1 -23173.861,E2 -23173.861} C_VEL
LIN {X 0,Y 209.998,Z 475.213,A -85,B 0,C 180,E1 -23177.418,E2 -23177.418} C_VEL
LIN {X 0,Y 220.588,Z 468.772,A -85,B 0,C 180,E1 -23179.878,E2 -23179.878} C_VEL
LIN {X 0,Y 224.461,Z 466.292,A -85,B 0,C 180,E1 -23180.637,E2 -23180.637} C_VEL
LIN {X 0,Y 224.002,Z 466.273,A -85,B 0,C 180,E1 -23181.135,E2 -23181.135} C_VEL
LIN {X 0,Y 214.006,Z 469.815,A -85,B 0,C 180,E1 -23183.763,E2 -23183.763} C_VEL
LIN {X 0,Y 204.665,Z 472.142,A -85,B 0,C 180,E1 -23186.673,E2 -23186.673} C_VEL
LIN {X 0,Y 196.094,Z 473.237,A -85,B 0,C 180,E1 -23189.884,E2 -23189.884} C_VEL
LIN {X 0,Y 188.376,Z 473.1,A -85,B 0,C 180,E1 -23193.404,E2 -23193.404} C_VEL
LIN {X 0,Y 181.483,Z 471.72,A -85,B 0,C 180,E1 -23197.217,E2 -23197.217} C_VEL
LIN {X 0,Y 175.817,Z 469.004,A -85,B 0,C 180,E1 -23201.35,E2 -23201.35} C_VEL
LIN {X 0,Y 171.146,Z 464.942,A -85,B 0,C 180,E1 -23205.736,E2 -23205.736} C_VEL
LIN {X 0,Y 167.939,Z 459.445,A -85,B 0,C 180,E1 -23210.364,E2 -23210.364} C_VEL
LIN {X 0,Y 165.573,Z 452.385,A -85,B 0,C 180,E1 -23215.13,E2 -23215.13} C_VEL
LIN {X 0,Y 164.443,Z 444.636,A -85,B 0,C 180,E1 -23219.388,E2 -23219.388} C_VEL
LIN {X 0,Y 164.143,Z 435.313,A -85,B 0,C 180,E1 -23223.683,E2 -23223.683} C_VEL
LIN {X 0,Y 164.396,Z 425.664,A -85,B 0,C 180,E1 -23227.369,E2 -23227.369} C_VEL
LIN {X 0,Y 165.024,Z 414.301,A -85,B 0,C 180,E1 -23231.003,E2 -23231.003} C_VEL
LIN {X 0,Y 165.913,Z 402.71,A -85,B 0,C 180,E1 -23234.097,E2 -23234.097} C_VEL
LIN {X 0,Y 166.106,Z 399.701,A -85,B 0,C 180,E1 -23234.863,E2 -23234.863} C_VEL
LIN {X 0,Y 166.201,Z 400.239,A -85,B 0,C 180,E1 -23235.325,E2 -23235.325} C_VEL
LIN {X 0,Y 166.671,Z 400.107,A -85,B 0,C 180,E1 -23235.908,E2 -23235.908} C_VEL
LIN {X 0,Y 168.097,Z 398.7,A -85,B 0,C 180,E1 -23237.018,E2 -23237.018} C_VEL
LIN {X 0,Y 170.092,Z 396.108,A -85,B 0,C 180,E1 -23238.125,E2 -23238.125} C_VEL
LIN {X 0,Y 173.325,Z 391.053,A -85,B 0,C 180,E1 -23239.544,E2 -23239.544} C_VEL
LIN {X 0,Y 174.004,Z 390.659,A -85,B 0,C 180,E1 -23240.079,E2 -23240.079} C_VEL
LIN {X 0,Y 175.671,Z 389.056,A -85,B 0,C 180,E1 -23241.104,E2 -23241.104} C_VEL
LIN {X 0,Y 178.952,Z 384.639,A -85,B 0,C 180,E1 -23242.607,E2 -23242.607} C_VEL
LIN {X 0,Y 182.536,Z 378.366,A -85,B 0,C 180,E1 -23243.846,E2 -23243.846} C_VEL
LIN {X 0,Y 184.138,Z 375.156,A -85,B 0,C 180,E1 -23244.374,E2 -23244.374} C_VEL
LIN {X 0,Y 186.562,Z 372.265,A -85,B 0,C 180,E1 -23245.516,E2 -23245.516} C_VEL
LIN {X 0,Y 189.704,Z 367.017,A -85,B 0,C 180,E1 -23246.711,E2 -23246.711} C_VEL
LIN {X 0,Y 192.959,Z 359.775,A -85,B 0,C 180,E1 -23247.744,E2 -23247.744} C_VEL
LIN {X 0,Y 196.095,Z 350.427,A -85,B 0,C 180,E1 -23248.644,E2 -23248.644} C_VEL
LIN {X 0,Y 198.499,Z 341.694,A -85,B 0,C 180,E1 -23249.278,E2 -23249.278} C_VEL
LIN {X 0,Y 201.367,Z 336.246,A -85,B 0,C 180,E1 -23250.35,E2 -23250.35} C_VEL
LIN {X 0,Y 204.057,Z 329.364,A -85,B 0,C 180,E1 -23251.178,E2 -23251.178} C_VEL
LIN {X 0,Y 208.284,Z 315.82,A -85,B 0,C 180,E1 -23252.224,E2 -23252.224} C_VEL
LIN {X 0,Y 211.522,Z 303.825,A -85,B 0,C 180,E1 -23252.877,E2 -23252.877} C_VEL
LIN {X 0,Y 214.686,Z 297.607,A -85,B 0,C 180,E1 -23253.815,E2 -23253.815} C_VEL
LIN {X 0,Y 218.15,Z 288.77,A -85,B 0,C 180,E1 -23254.67,E2 -23254.67} C_VEL
LIN {X 0,Y 222.741,Z 274.115,A -85,B 0,C 180,E1 -23255.574,E2 -23255.574} C_VEL
LIN {X 0,Y 225.295,Z 265.047,A -85,B 0,C 180,E1 -23256.003,E2 -23256.003} C_VEL
LIN {X 0,Y 225.56,Z 264.95,A -85,B 0,C 180,E1 -23256.092,E2 -23256.092} C_VEL
LIN {X 0,Y 226.6,Z 267.23,A -85,B 0,C 180,E1 -23256.578,E2 -23256.578} C_VEL
LIN {X 0,Y 220.046,Z 355.52,A -85,B 0,C 180,E1 -23259.055,E2 -23259.055} C_VEL
LIN {X 0,Y 218.165,Z 370.476,A -85,B 0,C 180,E1 -23259.781,E2 -23259.781} C_VEL
LIN {X 0,Y 215.714,Z 383.985,A -85,B 0,C 180,E1 -23260.713,E2 -23260.713} C_VEL
LIN {X 0,Y 212.676,Z 397.379,A -85,B 0,C 180,E1 -23261.964,E2 -23261.964} C_VEL
LIN {X 0,Y 208.588,Z 411.237,A -85,B 0,C 180,E1 -23263.578,E2 -23263.578} C_VEL
LIN {X 0,Y 204.067,Z 423.886,A -85,B 0,C 180,E1 -23265.433,E2 -23265.433} C_VEL
LIN {X 0,Y 198.643,Z 436.62,A -85,B 0,C 180,E1 -23267.758,E2 -23267.758} C_VEL
LIN {X 0,Y 193.276,Z 448.109,A -85,B 0,C 180,E1 -23270.477,E2 -23270.477} C_VEL
LIN {X 0,Y 188.332,Z 457.752,A -85,B 0,C 180,E1 -23273.336,E2 -23273.336} C_VEL
LIN {X 0,Y 182.859,Z 467.18,A -85,B 0,C 180,E1 -23276.789,E2 -23276.789} C_VEL
LIN {X 0,Y 177.82,Z 475.34,A -85,B 0,C 180,E1 -23280.61,E2 -23280.61} C_VEL
LIN {X 0,Y 173.393,Z 482.274,A -85,B 0,C 180,E1 -23284.809,E2 -23284.809} C_VEL
LIN {X 0,Y 169.576,Z 488.022,A -85,B 0,C 180,E1 -23289.37,E2 -23289.37} C_VEL
LIN {X 0,Y 167.388,Z 491.398,A -85,B 0,C 180,E1 -23292.905,E2 -23292.905} C_VEL
LIN {X 0,Y 165.153,Z 494.836,A -85,B 0,C 180,E1 -23297.712,E2 -23297.712} C_VEL
LIN {X 0,Y 163.728,Z 497.094,A -85,B 0,C 180,E1 -23302.598,E2 -23302.598} C_VEL
LIN {X 0,Y 163.156,Z 498.227,A -85,B 0,C 180,E1 -23307.528,E2 -23307.528} C_VEL
LIN {X 0,Y 163.154,Z 498.237,A -85,B 0,C 180,E1 -23312.466,E2 -23312.466} C_VEL
LIN {X 0,Y 163.717,Z 497.145,A -85,B 0,C 180,E1 -23317.396,E2 -23317.396} C_VEL
LIN {X 0,Y 165.151,Z 494.929,A -85,B 0,C 180,E1 -23322.282,E2 -23322.282} C_VEL
LIN {X 0,Y 167.331,Z 491.547,A -85,B 0,C 180,E1 -23327.094,E2 -23327.094} C_VEL
LIN {X 0,Y 170.39,Z 486.897,A -85,B 0,C 180,E1 -23331.787,E2 -23331.787} C_VEL
LIN {X 0,Y 174.419,Z 480.836,A -85,B 0,C 180,E1 -23336.307,E2 -23336.307} C_VEL
LIN {X 0,Y 179.235,Z 473.203,A -85,B 0,C 180,E1 -23340.643,E2 -23340.643} C_VEL
LIN {X 0,Y 184.249,Z 465.028,A -85,B 0,C 180,E1 -23344.234,E2 -23344.234} C_VEL
LIN {X 0,Y 189.043,Z 456.71,A -85,B 0,C 180,E1 -23347.162,E2 -23347.162} C_VEL
LIN {X 0,Y 194.029,Z 446.859,A -85,B 0,C 180,E1 -23350.007,E2 -23350.007} C_VEL
LIN {X 0,Y 199.064,Z 436.153,A -85,B 0,C 180,E1 -23352.467,E2 -23352.467} C_VEL
LIN {X 0,Y 203.981,Z 424.578,A -85,B 0,C 180,E1 -23354.584,E2 -23354.584} C_VEL
LIN {X 0,Y 208.473,Z 412.07,A -85,B 0,C 180,E1 -23356.448,E2 -23356.448} C_VEL
LIN {X 0,Y 212.57,Z 398.418,A -85,B 0,C 180,E1 -23358.06,E2 -23358.06} C_VEL
LIN {X 0,Y 216.062,Z 383.233,A -85,B 0,C 180,E1 -23359.475,E2 -23359.475} C_VEL
LIN {X 0,Y 218.664,Z 368.325,A -85,B 0,C 180,E1 -23360.473,E2 -23360.473} C_VEL
LIN {X 0,Y 220.506,Z 352.948,A -85,B 0,C 180,E1 -23361.153,E2 -23361.153} C_VEL
LIN {X 0,Y 224.978,Z 292.56,A -85,B 0,C 180,E1 -23362.84,E2 -23362.84} C_VEL
LIN {X 0,Y 226.798,Z 267.326,A -85,B 0,C 180,E1 -23363.54,E2 -23363.54} C_VEL
LIN {X 0,Y 221.121,Z 256.045,A -85,B 0,C 180,E1 -23366.265,E2 -23366.265} C_VEL
LIN {X 0,Y 215.916,Z 246.752,A -85,B 0,C 180,E1 -23369.023,E2 -23369.023} C_VEL
LIN {X 0,Y 211.711,Z 239.933,A -85,B 0,C 180,E1 -23371.491,E2 -23371.491} C_VEL
LIN {X 0,Y 207.313,Z 233.261,A -85,B 0,C 180,E1 -23374.39,E2 -23374.39} C_VEL
LIN {X 0,Y 204.36,Z 229.201,A -85,B 0,C 180,E1 -23376.569,E2 -23376.569} C_VEL
LIN {X 0,Y 201.409,Z 225.103,A -85,B 0,C 180,E1 -23379.043,E2 -23379.043} C_VEL
LIN {X 0,Y 198.183,Z 220.934,A -85,B 0,C 180,E1 -23382.19,E2 -23382.19} C_VEL
LIN {X 0,Y 194.459,Z 216.161,A -85,B 0,C 180,E1 -23386.9,E2 -23386.9} C_VEL
LIN {X 0,Y 191.01,Z 211.929,A -85,B 0,C 180,E1 -23394.457,E2 -23394.457} C_VEL
LIN {X 0,Y 190.466,Z 210.857,A -85,B 0,C 180,E1 -23397.885,E2 -23397.885} C_VEL
LIN {X 0,Y 190.493,Z 210.944,A -85,B 0,C 180,E1 -23401.585,E2 -23401.585} C_VEL
LIN {X 0,Y 193.622,Z 216.111,A -85,B 0,C 180,E1 -23411.052,E2 -23411.052} C_VEL
LIN {X 0,Y 197.776,Z 221.759,A -85,B 0,C 180,E1 -23416.645,E2 -23416.645} C_VEL
LIN {X 0,Y 201.461,Z 226.84,A -85,B 0,C 180,E1 -23420.284,E2 -23420.284} C_VEL
LIN {X 0,Y 204.95,Z 231.851,A -85,B 0,C 180,E1 -23423.158,E2 -23423.158} C_VEL
LIN {X 0,Y 209.531,Z 238.616,A -85,B 0,C 180,E1 -23426.386,E2 -23426.386} C_VEL
LIN {X 0,Y 215.33,Z 247.922,A -85,B 0,C 180,E1 -23429.899,E2 -23429.899} C_VEL
LIN {X 0,Y 217.818,Z 252.491,A -85,B 0,C 180,E1 -23431.281,E2 -23431.281} C_VEL
LIN {X 0,Y 222.494,Z 267.669,A -85,B 0,C 180,E1 -23434.034,E2 -23434.034} C_VEL
LIN {X 0,Y 223.931,Z 272.731,A -85,B 0,C 180,E1 -23434.842,E2 -23434.842} C_VEL
LIN {X 0,Y 224.126,Z 282.729,A -85,B 0,C 180,E1 -23435.45,E2 -23435.45} C_VEL
LIN {X 0,Y 223.701,Z 288.593,A -85,B 0,C 180,E1 -23435.613,E2 -23435.613} C_VEL
LIN {X 0,Y 221.802,Z 298.328,A -85,B 0,C 180,E1 -23435.463,E2 -23435.463} C_VEL
LIN {X 0,Y 220.048,Z 306.133,A -85,B 0,C 180,E1 -23435.257,E2 -23435.257} C_VEL
LIN {X 0,Y 219.086,Z 312.047,A -85,B 0,C 180,E1 -23435.231,E2 -23435.231} C_VEL
LIN {X 0,Y 218.897,Z 314.03,A -85,B 0,C 180,E1 -23435.271,E2 -23435.271} C_VEL
LIN {X 0,Y 213.826,Z 378.373,A -85,B 0,C 180,E1 -23437.058,E2 -23437.058} C_VEL
LIN {X 0,Y 211.513,Z 393.651,A -85,B 0,C 180,E1 -23437.705,E2 -23437.705} C_VEL
LIN {X 0,Y 208.421,Z 407.828,A -85,B 0,C 180,E1 -23438.571,E2 -23438.571} C_VEL
LIN {X 0,Y 204.42,Z 421.87,A -85,B 0,C 180,E1 -23439.717,E2 -23439.717} C_VEL
LIN {X 0,Y 199.649,Z 435.6,A -85,B 0,C 180,E1 -23441.203,E2 -23441.203} C_VEL
LIN {X 0,Y 194.452,Z 448.224,A -85,B 0,C 180,E1 -23442.96,E2 -23442.96} C_VEL
LIN {X 0,Y 189.168,Z 459.966,A -85,B 0,C 180,E1 -23445.103,E2 -23445.103} C_VEL
LIN {X 0,Y 183.046,Z 471.759,A -85,B 0,C 180,E1 -23447.79,E2 -23447.79} C_VEL
LIN {X 0,Y 177.473,Z 481.709,A -85,B 0,C 180,E1 -23450.687,E2 -23450.687} C_VEL
LIN {X 0,Y 171.712,Z 491.471,A -85,B 0,C 180,E1 -23454.325,E2 -23454.325} C_VEL
LIN {X 0,Y 167.417,Z 498.57,A -85,B 0,C 180,E1 -23457.644,E2 -23457.644} C_VEL
LIN {X 0,Y 163.173,Z 505.508,A -85,B 0,C 180,E1 -23461.724,E2 -23461.724} C_VEL
LIN {X 0,Y 159.388,Z 511.975,A -85,B 0,C 180,E1 -23466.623,E2 -23466.623} C_VEL
LIN {X 0,Y 156.849,Z 517.014,A -85,B 0,C 180,E1 -23471.724,E2 -23471.724} C_VEL
LIN {X 0,Y 155.427,Z 520.742,A -85,B 0,C 180,E1 -23476.937,E2 -23476.937} C_VEL
LIN {X 0,Y 155.186,Z 523.252,A -85,B 0,C 180,E1 -23482.195,E2 -23482.195} C_VEL
LIN {X 0,Y 155.442,Z 524.062,A -85,B 0,C 180,E1 -23484.815,E2 -23484.815} C_VEL
LIN {X 0,Y 155.958,Z 524.746,A -85,B 0,C 180,E1 -23490.003,E2 -23490.003} C_VEL
LIN {X 0,Y 155.509,Z 524.055,A -85,B 0,C 180,E1 -23495.189,E2 -23495.189} C_VEL
LIN {X 0,Y 155.211,Z 522.117,A -85,B 0,C 180,E1 -23500.438,E2 -23500.438} C_VEL
LIN {X 0,Y 156.038,Z 518.981,A -85,B 0,C 180,E1 -23505.682,E2 -23505.682} C_VEL
LIN {X 0,Y 157.937,Z 514.575,A -85,B 0,C 180,E1 -23510.857,E2 -23510.857} C_VEL
LIN {X 0,Y 161.144,Z 508.821,A -85,B 0,C 180,E1 -23515.861,E2 -23515.861} C_VEL
LIN {X 0,Y 165.507,Z 501.556,A -85,B 0,C 180,E1 -23520.638,E2 -23520.638} C_VEL
LIN {X 0,Y 170.327,Z 493.641,A -85,B 0,C 180,E1 -23524.662,E2 -23524.662} C_VEL
LIN {X 0,Y 172.445,Z 490.592,A -85,B 0,C 180,E1 -23526.047,E2 -23526.047} C_VEL
LIN {X 0,Y 181.867,Z 486.879,A -85,B 0,C 180,E1 -23531.07,E2 -23531.07} C_VEL
LIN {X 0,Y 192.745,Z 482.061,A -85,B 0,C 180,E1 -23535.321,E2 -23535.321} C_VEL
LIN {X 0,Y 205.302,Z 475.963,A -85,B 0,C 180,E1 -23538.864,E2 -23538.864} C_VEL
LIN {X 0,Y 212.662,Z 472.017,A -85,B 0,C 180,E1 -23540.574,E2 -23540.574} C_VEL
LIN {X 0,Y 213.732,Z 471.112,A -85,B 0,C 180,E1 -23541.335,E2 -23541.335} C_VEL
LIN {X 0,Y 203.761,Z 473.525,A -85,B 0,C 180,E1 -23544.102,E2 -23544.102} C_VEL
LIN {X 0,Y 194.478,Z 474.775,A -85,B 0,C 180,E1 -23547.176,E2 -23547.176} C_VEL
LIN {X 0,Y 186.046,Z 474.807,A -85,B 0,C 180,E1 -23550.589,E2 -23550.589} C_VEL
LIN {X 0,Y 178.489,Z 473.621,A -85,B 0,C 180,E1 -23554.334,E2 -23554.334} C_VEL
LIN {X 0,Y 171.883,Z 471.173,A -85,B 0,C 180,E1 -23558.408,E2 -23558.408} C_VEL
LIN {X 0,Y 166.497,Z 467.397,A -85,B 0,C 180,E1 -23562.814,E2 -23562.814} C_VEL
LIN {X 0,Y 162.484,Z 462.197,A -85,B 0,C 180,E1 -23567.51,E2 -23567.51} C_VEL
LIN {X 0,Y 160.217,Z 457.357,A -85,B 0,C 180,E1 -23571.169,E2 -23571.169} C_VEL
LIN {X 0,Y 158.312,Z 450.48,A -85,B 0,C 180,E1 -23575.545,E2 -23575.545} C_VEL
LIN {X 0,Y 157.309,Z 442.144,A -85,B 0,C 180,E1 -23580,E2 -23580} C_VEL
LIN {X 0,Y 157.088,Z 432.026,A -85,B 0,C 180,E1 -23584.491,E2 -23584.491} C_VEL
LIN {X 0,Y 157.511,Z 421.7,A -85,B 0,C 180,E1 -23588.338,E2 -23588.338} C_VEL
LIN {X 0,Y 158.014,Z 412.96,A -85,B 0,C 180,E1 -23591.106,E2 -23591.106} C_VEL
LIN {X 0,Y 158.011,Z 413.298,A -85,B 0,C 180,E1 -23591.498,E2 -23591.498} C_VEL
LIN {X 0,Y 158.843,Z 412.869,A -85,B 0,C 180,E1 -23592.781,E2 -23592.781} C_VEL
LIN {X 0,Y 161.078,Z 410.433,A -85,B 0,C 180,E1 -23594.53,E2 -23594.53} C_VEL
LIN {X 0,Y 163.96,Z 406.639,A -85,B 0,C 180,E1 -23596.178,E2 -23596.178} C_VEL
LIN {X 0,Y 165.221,Z 405.781,A -85,B 0,C 180,E1 -23597.323,E2 -23597.323} C_VEL
LIN {X 0,Y 166.907,Z 404.22,A -85,B 0,C 180,E1 -23598.484,E2 -23598.484} C_VEL
LIN {X 0,Y 169.876,Z 400.66,A -85,B 0,C 180,E1 -23599.957,E2 -23599.957} C_VEL
LIN {X 0,Y 172.294,Z 397.191,A -85,B 0,C 180,E1 -23600.911,E2 -23600.911} C_VEL
LIN {X 0,Y 174.733,Z 395.033,A -85,B 0,C 180,E1 -23602.311,E2 -23602.311} C_VEL
LIN {X 0,Y 178.199,Z 390.94,A -85,B 0,C 180,E1 -23603.844,E2 -23603.844} C_VEL
LIN {X 0,Y 181.997,Z 385.415,A -85,B 0,C 180,E1 -23605.137,E2 -23605.137} C_VEL
LIN {X 0,Y 184.91,Z 380.278,A -85,B 0,C 180,E1 -23605.986,E2 -23605.986} C_VEL
LIN {X 0,Y 188.056,Z 376.506,A -85,B 0,C 180,E1 -23607.246,E2 -23607.246} C_VEL
LIN {X 0,Y 191.742,Z 370.575,A -85,B 0,C 180,E1 -23608.457,E2 -23608.457} C_VEL
LIN {X 0,Y 195.469,Z 362.804,A -85,B 0,C 180,E1 -23609.488,E2 -23609.488} C_VEL
LIN {X 0,Y 199.129,Z 352.586,A -85,B 0,C 180,E1 -23610.396,E2 -23610.396} C_VEL
LIN {X 0,Y 201.264,Z 345.289,A -85,B 0,C 180,E1 -23610.929,E2 -23610.929} C_VEL
LIN {X 0,Y 204.209,Z 339.576,A -85,B 0,C 180,E1 -23611.932,E2 -23611.932} C_VEL
LIN {X 0,Y 207.094,Z 332.374,A -85,B 0,C 180,E1 -23612.758,E2 -23612.758} C_VEL
LIN {X 0,Y 211.603,Z 318.266,A -85,B 0,C 180,E1 -23613.797,E2 -23613.797} C_VEL
LIN {X 0,Y 214.736,Z 307.104,A -85,B 0,C 180,E1 -23614.399,E2 -23614.399} C_VEL
LIN {X 0,Y 218.107,Z 300.4,A -85,B 0,C 180,E1 -23615.317,E2 -23615.317} C_VEL
LIN {X 0,Y 220.294,Z 295.024,A -85,B 0,C 180,E1 -23615.83,E2 -23615.83} C_VEL
LIN {X 0,Y 215.666,Z 356.042,A -85,B 0,C 180,E1 -23617.598,E2 -23617.598} C_VEL
LIN {X 0,Y 213.693,Z 371.137,A -85,B 0,C 180,E1 -23618.33,E2 -23618.33} C_VEL
LIN {X 0,Y 211.087,Z 384.948,A -85,B 0,C 180,E1 -23619.292,E2 -23619.292} C_VEL
LIN {X 0,Y 208.021,Z 397.947,A -85,B 0,C 180,E1 -23620.518,E2 -23620.518} C_VEL
LIN {X 0,Y 203.785,Z 411.811,A -85,B 0,C 180,E1 -23622.139,E2 -23622.139} C_VEL
LIN {X 0,Y 199.088,Z 424.464,A -85,B 0,C 180,E1 -23624.004,E2 -23624.004} C_VEL
LIN {X 0,Y 193.457,Z 437.201,A -85,B 0,C 180,E1 -23626.348,E2 -23626.348} C_VEL
LIN {X 0,Y 187.865,Z 448.692,A -85,B 0,C 180,E1 -23629.102,E2 -23629.102} C_VEL
LIN {X 0,Y 182.697,Z 458.336,A -85,B 0,C 180,E1 -23632.009,E2 -23632.009} C_VEL
LIN {X 0,Y 176.964,Z 467.766,A -85,B 0,C 180,E1 -23635.53,E2 -23635.53} C_VEL
LIN {X 0,Y 171.504,Z 476.174,A -85,B 0,C 180,E1 -23639.587,E2 -23639.587} C_VEL
LIN {X 0,Y 167.022,Z 482.858,A -85,B 0,C 180,E1 -23643.777,E2 -23643.777} C_VEL
LIN {X 0,Y 162.967,Z 488.607,A -85,B 0,C 180,E1 -23648.493,E2 -23648.493} C_VEL
LIN {X 0,Y 160.616,Z 491.985,A -85,B 0,C 180,E1 -23652.161,E2 -23652.161} C_VEL
LIN {X 0,Y 158.229,Z 495.422,A -85,B 0,C 180,E1 -23657.165,E2 -23657.165} C_VEL
LIN {X 0,Y 156.722,Z 497.679,A -85,B 0,C 180,E1 -23662.265,E2 -23662.265} C_VEL
LIN {X 0,Y 156.085,Z 498.812,A -85,B 0,C 180,E1 -23667.416,E2 -23667.416} C_VEL
LIN {X 0,Y 156.082,Z 498.822,A -85,B 0,C 180,E1 -23672.577,E2 -23672.577} C_VEL
LIN {X 0,Y 156.712,Z 497.728,A -85,B 0,C 180,E1 -23677.729,E2 -23677.729} C_VEL
LIN {X 0,Y 158.226,Z 495.514,A -85,B 0,C 180,E1 -23682.828,E2 -23682.828} C_VEL
LIN {X 0,Y 160.569,Z 492.132,A -85,B 0,C 180,E1 -23687.838,E2 -23687.838} C_VEL
LIN {X 0,Y 163.831,Z 487.481,A -85,B 0,C 180,E1 -23692.707,E2 -23692.707} C_VEL
LIN {X 0,Y 168.104,Z 481.418,A -85,B 0,C 180,E1 -23697.376,E2 -23697.376} C_VEL
LIN {X 0,Y 173.172,Z 473.785,A -85,B 0,C 180,E1 -23701.839,E2 -23701.839} C_VEL
LIN {X 0,Y 178.44,Z 465.608,A -85,B 0,C 180,E1 -23705.513,E2 -23705.513} C_VEL
LIN {X 0,Y 183.446,Z 457.289,A -85,B 0,C 180,E1 -23708.499,E2 -23708.499} C_VEL
LIN {X 0,Y 188.651,Z 447.437,A -85,B 0,C 180,E1 -23711.392,E2 -23711.392} C_VEL
LIN {X 0,Y 193.904,Z 436.727,A -85,B 0,C 180,E1 -23713.878,E2 -23713.878} C_VEL
LIN {X 0,Y 199.003,Z 425.148,A -85,B 0,C 180,E1 -23716.014,E2 -23716.014} C_VEL
LIN {X 0,Y 203.677,Z 412.633,A -85,B 0,C 180,E1 -23717.887,E2 -23717.887} C_VEL
LIN {X 0,Y 207.914,Z 398.976,A -85,B 0,C 180,E1 -23719.509,E2 -23719.509} C_VEL
LIN {X 0,Y 211.447,Z 384.207,A -85,B 0,C 180,E1 -23720.896,E2 -23720.896} C_VEL
LIN {X 0,Y 214.163,Z 369.331,A -85,B 0,C 180,E1 -23721.903,E2 -23721.903} C_VEL
LIN {X 0,Y 216.014,Z 354.824,A -85,B 0,C 180,E1 -23722.562,E2 -23722.562} C_VEL
LIN {X 0,Y 220.782,Z 293.014,A -85,B 0,C 180,E1 -23724.301,E2 -23724.301} C_VEL
LIN {X 0,Y 222.471,Z 270.41,A -85,B 0,C 180,E1 -23724.931,E2 -23724.931} C_VEL
LIN {X 0,Y 217.757,Z 260.791,A -85,B 0,C 180,E1 -23727.349,E2 -23727.349} C_VEL
LIN {X 0,Y 213.036,Z 252.143,A -85,B 0,C 180,E1 -23730,E2 -23730} C_VEL
LIN {X 0,Y 209.063,Z 245.496,A -85,B 0,C 180,E1 -23732.469,E2 -23732.469} C_VEL
LIN {X 0,Y 204.69,Z 238.745,A -85,B 0,C 180,E1 -23735.533,E2 -23735.533} C_VEL
LIN {X 0,Y 201.886,Z 234.792,A -85,B 0,C 180,E1 -23737.754,E2 -23737.754} C_VEL
LIN {X 0,Y 199.629,Z 231.538,A -85,B 0,C 180,E1 -23739.773,E2 -23739.773} C_VEL
LIN {X 0,Y 196.508,Z 227.362,A -85,B 0,C 180,E1 -23742.998,E2 -23742.998} C_VEL
LIN {X 0,Y 193.399,Z 223.155,A -85,B 0,C 180,E1 -23747.139,E2 -23747.139} C_VEL
LIN {X 0,Y 190.079,Z 218.924,A -85,B 0,C 180,E1 -23754.696,E2 -23754.696} C_VEL
LIN {X 0,Y 189.601,Z 217.906,A -85,B 0,C 180,E1 -23757.875,E2 -23757.875} C_VEL
LIN {X 0,Y 189.585,Z 217.898,A -85,B 0,C 180,E1 -23761.062,E2 -23761.062} C_VEL
LIN {X 0,Y 191.361,Z 221.623,A -85,B 0,C 180,E1 -23768.447,E2 -23768.447} C_VEL
LIN {X 0,Y 193.01,Z 223.8,A -85,B 0,C 180,E1 -23771.552,E2 -23771.552} C_VEL
LIN {X 0,Y 196.351,Z 228.49,A -85,B 0,C 180,E1 -23776.105,E2 -23776.105} C_VEL
LIN {X 0,Y 199.722,Z 233.291,A -85,B 0,C 180,E1 -23779.596,E2 -23779.596} C_VEL
LIN {X 0,Y 203.461,Z 238.852,A -85,B 0,C 180,E1 -23782.8,E2 -23782.8} C_VEL
LIN {X 0,Y 208.115,Z 246.103,A -85,B 0,C 180,E1 -23786.175,E2 -23786.175} C_VEL
LIN {X 0,Y 213.218,Z 254.583,A -85,B 0,C 180,E1 -23789.359,E2 -23789.359} C_VEL
LIN {X 0,Y 214.772,Z 257.744,A -85,B 0,C 180,E1 -23790.278,E2 -23790.278} C_VEL
LIN {X 0,Y 219.792,Z 275.056,A -85,B 0,C 180,E1 -23793.421,E2 -23793.421} C_VEL
LIN {X 0,Y 220.185,Z 295.76,A -85,B 0,C 180,E1 -23794.736,E2 -23794.736} C_VEL
LIN {X 0,Y 218.897,Z 314.03,A -85,B 0,C 180,E1 -23795.271,E2 -23795.271} C_VEL
LIN {X 0,Y 218.067,Z 319.88,A -85,B 0,C 180,E1 -23795.291,E2 -23795.291} C_VEL
LIN {X 0,Y 213.225,Z 338.931,A -85,B 0,C 180,E1 -23794.551,E2 -23794.551} C_VEL
LIN {X 0,Y 212.367,Z 344.783,A -85,B 0,C 180,E1 -23794.558,E2 -23794.558} C_VEL
LIN {X 0,Y 209.48,Z 379.228,A -85,B 0,C 180,E1 -23795.558,E2 -23795.558} C_VEL
LIN {X 0,Y 206.919,Z 394.79,A -85,B 0,C 180,E1 -23796.233,E2 -23796.233} C_VEL
LIN {X 0,Y 203.441,Z 409.74,A -85,B 0,C 180,E1 -23797.188,E2 -23797.188} C_VEL
LIN {X 0,Y 199.322,Z 423.266,A -85,B 0,C 180,E1 -23798.328,E2 -23798.328} C_VEL
LIN {X 0,Y 194.44,Z 436.603,A -85,B 0,C 180,E1 -23799.823,E2 -23799.823} C_VEL
LIN {X 0,Y 188.522,Z 450.224,A -85,B 0,C 180,E1 -23801.795,E2 -23801.795} C_VEL
LIN {X 0,Y 182.566,Z 462.595,A -85,B 0,C 180,E1 -23804.199,E2 -23804.199} C_VEL
LIN {X 0,Y 175.784,Z 474.71,A -85,B 0,C 180,E1 -23807.186,E2 -23807.186} C_VEL
LIN {X 0,Y 170.17,Z 484.12,A -85,B 0,C 180,E1 -23810.202,E2 -23810.202} C_VEL
LIN {X 0,Y 164.333,Z 493.366,A -85,B 0,C 180,E1 -23813.98,E2 -23813.98} C_VEL
LIN {X 0,Y 159.33,Z 501.093,A -85,B 0,C 180,E1 -23818.045,E2 -23818.045} C_VEL
LIN {X 0,Y 154.676,Z 508.336,A -85,B 0,C 180,E1 -23822.98,E2 -23822.98} C_VEL
LIN {X 0,Y 151.122,Z 514.33,A -85,B 0,C 180,E1 -23828.451,E2 -23828.451} C_VEL
LIN {X 0,Y 149.098,Z 518.443,A -85,B 0,C 180,E1 -23833.575,E2 -23833.575} C_VEL
LIN {X 0,Y 148.132,Z 521.554,A -85,B 0,C 180,E1 -23839.064,E2 -23839.064} C_VEL
LIN {X 0,Y 148.342,Z 523.473,A -85,B 0,C 180,E1 -23844.566,E2 -23844.566} C_VEL
LIN {X 0,Y 148.865,Z 524.159,A -85,B 0,C 180,E1 -23850.003,E2 -23850.003} C_VEL
LIN {X 0,Y 148.413,Z 523.465,A -85,B 0,C 180,E1 -23855.438,E2 -23855.438} C_VEL
LIN {X 0,Y 148.165,Z 521.524,A -85,B 0,C 180,E1 -23860.941,E2 -23860.941} C_VEL
LIN {X 0,Y 149.11,Z 518.385,A -85,B 0,C 180,E1 -23866.431,E2 -23866.431} C_VEL
LIN {X 0,Y 151.247,Z 513.981,A -85,B 0,C 180,E1 -23871.826,E2 -23871.826} C_VEL
LIN {X 0,Y 154.693,Z 508.226,A -85,B 0,C 180,E1 -23877.025,E2 -23877.025} C_VEL
LIN {X 0,Y 159.339,Z 500.96,A -85,B 0,C 180,E1 -23881.961,E2 -23881.961} C_VEL
LIN {X 0,Y 164.318,Z 493.295,A -85,B 0,C 180,E1 -23885.974,E2 -23885.974} C_VEL
LIN {X 0,Y 166.977,Z 489.519,A -85,B 0,C 180,E1 -23887.615,E2 -23887.615} C_VEL
LIN {X 0,Y 176.556,Z 486.335,A -85,B 0,C 180,E1 -23892.59,E2 -23892.59} C_VEL
LIN {X 0,Y 185.448,Z 482.989,A -85,B 0,C 180,E1 -23896.062,E2 -23896.062} C_VEL
LIN {X 0,Y 192.808,Z 479.99,A -85,B 0,C 180,E1 -23898.355,E2 -23898.355} C_VEL
LIN {X 0,Y 200.717,Z 476.524,A -85,B 0,C 180,E1 -23900.386,E2 -23900.386} C_VEL
LIN {X 0,Y 203.342,Z 474.99,A -85,B 0,C 180,E1 -23901.529,E2 -23901.529} C_VEL
LIN {X 0,Y 193.401,Z 476.322,A -85,B 0,C 180,E1 -23904.45,E2 -23904.45} C_VEL
LIN {X 0,Y 184.228,Z 476.502,A -85,B 0,C 180,E1 -23907.719,E2 -23907.719} C_VEL
LIN {X 0,Y 175.953,Z 475.48,A -85,B 0,C 180,E1 -23911.36,E2 -23911.36} C_VEL
LIN {X 0,Y 168.572,Z 473.229,A -85,B 0,C 180,E1 -23915.36,E2 -23915.36} C_VEL
LIN {X 0,Y 162.445,Z 469.69,A -85,B 0,C 180,E1 -23919.751,E2 -23919.751} C_VEL
LIN {X 0,Y 157.454,Z 464.817,A -85,B 0,C 180,E1 -23924.466,E2 -23924.466} C_VEL
LIN {X 0,Y 153.959,Z 458.503,A -85,B 0,C 180,E1 -23929.479,E2 -23929.479} C_VEL
LIN {X 0,Y 151.485,Z 450.527,A -85,B 0,C 180,E1 -23934.676,E2 -23934.676} C_VEL
LIN {X 0,Y 150.291,Z 440.662,A -85,B 0,C 180,E1 -23940,E2 -23940} C_VEL
LIN {X 0,Y 150.081,Z 431.719,A -85,B 0,C 180,E1 -23944.028,E2 -23944.028} C_VEL
LIN {X 0,Y 150.284,Z 424.802,A -85,B 0,C 180,E1 -23946.799,E2 -23946.799} C_VEL
LIN {X 0,Y 150.272,Z 425.037,A -85,B 0,C 180,E1 -23947.39,E2 -23947.39} C_VEL
LIN {X 0,Y 151.38,Z 423.999,A -85,B 0,C 180,E1 -23949.352,E2 -23949.352} C_VEL
LIN {X 0,Y 152.694,Z 422.448,A -85,B 0,C 180,E1 -23950.609,E2 -23950.609} C_VEL
LIN {X 0,Y 154.26,Z 420.507,A -85,B 0,C 180,E1 -23951.746,E2 -23951.746} C_VEL
LIN {X 0,Y 156.782,Z 418.305,A -85,B 0,C 180,E1 -23954.274,E2 -23954.274} C_VEL
LIN {X 0,Y 159.208,Z 415.863,A -85,B 0,C 180,E1 -23956.016,E2 -23956.016} C_VEL
LIN {X 0,Y 162.214,Z 412.389,A -85,B 0,C 180,E1 -23957.655,E2 -23957.655} C_VEL
LIN {X 0,Y 163.518,Z 411.474,A -85,B 0,C 180,E1 -23958.675,E2 -23958.675} C_VEL
LIN {X 0,Y 165.416,Z 409.862,A -85,B 0,C 180,E1 -23959.871,E2 -23959.871} C_VEL
LIN {X 0,Y 169.808,Z 404.956,A -85,B 0,C 180,E1 -23961.87,E2 -23961.87} C_VEL
LIN {X 0,Y 171.994,Z 402.276,A -85,B 0,C 180,E1 -23962.686,E2 -23962.686} C_VEL
LIN {X 0,Y 175.225,Z 399.387,A -85,B 0,C 180,E1 -23964.275,E2 -23964.275} C_VEL
LIN {X 0,Y 178.763,Z 395.331,A -85,B 0,C 180,E1 -23965.624,E2 -23965.624} C_VEL
LIN {X 0,Y 182.645,Z 390.085,A -85,B 0,C 180,E1 -23966.819,E2 -23966.819} C_VEL
LIN {X 0,Y 185.756,Z 385.194,A -85,B 0,C 180,E1 -23967.612,E2 -23967.612} C_VEL
LIN {X 0,Y 189.62,Z 380.569,A -85,B 0,C 180,E1 -23968.983,E2 -23968.983} C_VEL
LIN {X 0,Y 193.9,Z 374.039,A -85,B 0,C 180,E1 -23970.198,E2 -23970.198} C_VEL
LIN {X 0,Y 198.048,Z 365.881,A -85,B 0,C 180,E1 -23971.189,E2 -23971.189} C_VEL
LIN {X 0,Y 201.601,Z 356.826,A -85,B 0,C 180,E1 -23971.96,E2 -23971.96} C_VEL
LIN {X 0,Y 204.201,Z 348.787,A -85,B 0,C 180,E1 -23972.532,E2 -23972.532} C_VEL
LIN {X 0,Y 207.296,Z 342.724,A -85,B 0,C 180,E1 -23973.498,E2 -23973.498} C_VEL
LIN {X 0,Y 210.645,Z 334.372,A -85,B 0,C 180,E1 -23974.378,E2 -23974.378} C_VEL
LIN {X 0,Y 214.072,Z 324.011,A -85,B 0,C 180,E1 -23975.125,E2 -23975.125} C_VEL
LIN {X 0,Y 211.25,Z 358.395,A -85,B 0,C 180,E1 -23976.147,E2 -23976.147} C_VEL
LIN {X 0,Y 208.976,Z 374.245,A -85,B 0,C 180,E1 -23976.967,E2 -23976.967} C_VEL
LIN {X 0,Y 205.981,Z 388.865,A -85,B 0,C 180,E1 -23978.064,E2 -23978.064} C_VEL
LIN {X 0,Y 202.424,Z 402.36,A -85,B 0,C 180,E1 -23979.418,E2 -23979.418} C_VEL
LIN {X 0,Y 197.988,Z 415.459,A -85,B 0,C 180,E1 -23981.031,E2 -23981.031} C_VEL
LIN {X 0,Y 193.221,Z 427.547,A -85,B 0,C 180,E1 -23982.942,E2 -23982.942} C_VEL
LIN {X 0,Y 188.398,Z 437.781,A -85,B 0,C 180,E1 -23984.861,E2 -23984.861} C_VEL
LIN {X 0,Y 182.558,Z 449.276,A -85,B 0,C 180,E1 -23987.643,E2 -23987.643} C_VEL
LIN {X 0,Y 177.172,Z 458.919,A -85,B 0,C 180,E1 -23990.6,E2 -23990.6} C_VEL
LIN {X 0,Y 171.169,Z 468.35,A -85,B 0,C 180,E1 -23994.188,E2 -23994.188} C_VEL
LIN {X 0,Y 166.035,Z 475.897,A -85,B 0,C 180,E1 -23997.841,E2 -23997.841} C_VEL
LIN {X 0,Y 161.93,Z 481.762,A -85,B 0,C 180,E1 -24001.48,E2 -24001.48} C_VEL
LIN {X 0,Y 157.376,Z 487.87,A -85,B 0,C 180,E1 -24006.299,E2 -24006.299} C_VEL
LIN {X 0,Y 153.888,Z 492.571,A -85,B 0,C 180,E1 -24011.353,E2 -24011.353} C_VEL
LIN {X 0,Y 151.346,Z 496.007,A -85,B 0,C 180,E1 -24016.571,E2 -24016.571} C_VEL
LIN {X 0,Y 149.724,Z 498.263,A -85,B 0,C 180,E1 -24021.901,E2 -24021.901} C_VEL
LIN {X 0,Y 149.014,Z 499.397,A -85,B 0,C 180,E1 -24027.293,E2 -24027.293} C_VEL
LIN {X 0,Y 149.011,Z 499.407,A -85,B 0,C 180,E1 -24032.7,E2 -24032.7} C_VEL
LIN {X 0,Y 149.714,Z 498.312,A -85,B 0,C 180,E1 -24038.092,E2 -24038.092} C_VEL
LIN {X 0,Y 151.341,Z 496.097,A -85,B 0,C 180,E1 -24043.422,E2 -24043.422} C_VEL
LIN {X 0,Y 153.843,Z 492.715,A -85,B 0,C 180,E1 -24048.646,E2 -24048.646} C_VEL
LIN {X 0,Y 157.318,Z 488.064,A -85,B 0,C 180,E1 -24053.704,E2 -24053.704} C_VEL
LIN {X 0,Y 161.849,Z 482,A -85,B 0,C 180,E1 -24058.528,E2 -24058.528} C_VEL
LIN {X 0,Y 167.198,Z 474.366,A -85,B 0,C 180,E1 -24063.119,E2 -24063.119} C_VEL
LIN {X 0,Y 172.721,Z 466.188,A -85,B 0,C 180,E1 -24066.878,E2 -24066.878} C_VEL
LIN {X 0,Y 178.845,Z 456.305,A -85,B 0,C 180,E1 -24070.416,E2 -24070.416} C_VEL
LIN {X 0,Y 184.366,Z 446.203,A -85,B 0,C 180,E1 -24073.322,E2 -24073.322} C_VEL
LIN {X 0,Y 189.923,Z 435.188,A -85,B 0,C 180,E1 -24075.8,E2 -24075.8} C_VEL
LIN {X 0,Y 195.225,Z 423.2,A -85,B 0,C 180,E1 -24077.94,E2 -24077.94} C_VEL
LIN {X 0,Y 199.568,Z 411.659,A -85,B 0,C 180,E1 -24079.596,E2 -24079.596} C_VEL
LIN {X 0,Y 203.901,Z 397.715,A -85,B 0,C 180,E1 -24081.22,E2 -24081.22} C_VEL
LIN {X 0,Y 207.267,Z 383.803,A -85,B 0,C 180,E1 -24082.492,E2 -24082.492} C_VEL
LIN {X 0,Y 209.968,Z 369.376,A -85,B 0,C 180,E1 -24083.444,E2 -24083.444} C_VEL
LIN {X 0,Y 211.932,Z 353.917,A -85,B 0,C 180,E1 -24084.129,E2 -24084.129} C_VEL
LIN {X 0,Y 216.731,Z 293.463,A -85,B 0,C 180,E1 -24085.82,E2 -24085.82} C_VEL
LIN {X 0,Y 218.258,Z 273.374,A -85,B 0,C 180,E1 -24086.391,E2 -24086.391} C_VEL
LIN {X 0,Y 213.196,Z 263.041,A -85,B 0,C 180,E1 -24089.204,E2 -24089.204} C_VEL
LIN {X 0,Y 208.243,Z 253.947,A -85,B 0,C 180,E1 -24092.283,E2 -24092.283} C_VEL
LIN {X 0,Y 203.271,Z 245.861,A -85,B 0,C 180,E1 -24095.827,E2 -24095.827} C_VEL
LIN {X 0,Y 200.178,Z 241.313,A -85,B 0,C 180,E1 -24098.368,E2 -24098.368} C_VEL
LIN {X 0,Y 197.912,Z 237.997,A -85,B 0,C 180,E1 -24100.488,E2 -24100.488} C_VEL
LIN {X 0,Y 195.229,Z 234.228,A -85,B 0,C 180,E1 -24103.397,E2 -24103.397} C_VEL
LIN {X 0,Y 192.249,Z 230.04,A -85,B 0,C 180,E1 -24107.531,E2 -24107.531} C_VEL
LIN {X 0,Y 189.151,Z 225.919,A -85,B 0,C 180,E1 -24114.937,E2 -24114.937} C_VEL
LIN {X 0,Y 188.735,Z 224.963,A -85,B 0,C 180,E1 -24117.866,E2 -24117.866} C_VEL
LIN {X 0,Y 188.718,Z 224.963,A -85,B 0,C 180,E1 -24121.067,E2 -24121.067} C_VEL
LIN {X 0,Y 191.267,Z 229.731,A -85,B 0,C 180,E1 -24130.051,E2 -24130.051} C_VEL
LIN {X 0,Y 194.869,Z 235.066,A -85,B 0,C 180,E1 -24135.459,E2 -24135.459} C_VEL
LIN {X 0,Y 198.133,Z 239.959,A -85,B 0,C 180,E1 -24139.019,E2 -24139.019} C_VEL
LIN {X 0,Y 202.344,Z 246.433,A -85,B 0,C 180,E1 -24142.731,E2 -24142.731} C_VEL
LIN {X 0,Y 206.453,Z 253.197,A -85,B 0,C 180,E1 -24145.791,E2 -24145.791} C_VEL
LIN {X 0,Y 210.96,Z 261.064,A -85,B 0,C 180,E1 -24148.717,E2 -24148.717} C_VEL
LIN {X 0,Y 211.736,Z 262.991,A -85,B 0,C 180,E1 -24149.22,E2 -24149.22} C_VEL
LIN {X 0,Y 215.874,Z 277.956,A -85,B 0,C 180,E1 -24152.015,E2 -24152.015} C_VEL
LIN {X 0,Y 216.1,Z 297.295,A -85,B 0,C 180,E1 -24153.259,E2 -24153.259} C_VEL
LIN {X 0,Y 212.367,Z 344.783,A -85,B 0,C 180,E1 -24154.558,E2 -24154.558} C_VEL
LIN {X 0,Y 211.521,Z 350.636,A -85,B 0,C 180,E1 -24154.563,E2 -24154.563} C_VEL
LIN {X 0,Y 206.695,Z 369.677,A -85,B 0,C 180,E1 -24153.784,E2 -24153.784} C_VEL
LIN {X 0,Y 205.757,Z 375.506,A -85,B 0,C 180,E1 -24153.827,E2 -24153.827} C_VEL
LIN {X 0,Y 203.443,Z 390.807,A -85,B 0,C 180,E1 -24154.44,E2 -24154.44} C_VEL
LIN {X 0,Y 200.166,Z 405.448,A -85,B 0,C 180,E1 -24155.286,E2 -24155.286} C_VEL
LIN {X 0,Y 196.277,Z 418.787,A -85,B 0,C 180,E1 -24156.332,E2 -24156.332} C_VEL
LIN {X 0,Y 191.185,Z 432.891,A -85,B 0,C 180,E1 -24157.787,E2 -24157.787} C_VEL
LIN {X 0,Y 185.618,Z 445.788,A -85,B 0,C 180,E1 -24159.52,E2 -24159.52} C_VEL
LIN {X 0,Y 179.822,Z 457.738,A -85,B 0,C 180,E1 -24161.637,E2 -24161.637} C_VEL
LIN {X 0,Y 173.768,Z 468.803,A -85,B 0,C 180,E1 -24164.124,E2 -24164.124} C_VEL
LIN {X 0,Y 167.548,Z 479.026,A -85,B 0,C 180,E1 -24167.034,E2 -24167.034} C_VEL
LIN {X 0,Y 161.114,Z 489.042,A -85,B 0,C 180,E1 -24170.769,E2 -24170.769} C_VEL
LIN {X 0,Y 154.672,Z 498.444,A -85,B 0,C 180,E1 -24175.395,E2 -24175.395} C_VEL
LIN {X 0,Y 149.432,Z 506.086,A -85,B 0,C 180,E1 -24180.412,E2 -24180.412} C_VEL
LIN {X 0,Y 145.366,Z 512.186,A -85,B 0,C 180,E1 -24185.74,E2 -24185.74} C_VEL
LIN {X 0,Y 142.676,Z 516.908,A -85,B 0,C 180,E1 -24191.33,E2 -24191.33} C_VEL
LIN {X 0,Y 141.449,Z 519.554,A -85,B 0,C 180,E1 -24195.619,E2 -24195.619} C_VEL
LIN {X 0,Y 140.989,Z 522.067,A -85,B 0,C 180,E1 -24201.403,E2 -24201.403} C_VEL
LIN {X 0,Y 141.259,Z 522.885,A -85,B 0,C 180,E1 -24204.293,E2 -24204.293} C_VEL
LIN {X 0,Y 141.772,Z 523.573,A -85,B 0,C 180,E1 -24210.004,E2 -24210.004} C_VEL
LIN {X 0,Y 141.301,Z 522.875,A -85,B 0,C 180,E1 -24215.713,E2 -24215.713} C_VEL
LIN {X 0,Y 141.111,Z 520.93,A -85,B 0,C 180,E1 -24221.495,E2 -24221.495} C_VEL
LIN {X 0,Y 142.22,Z 517.79,A -85,B 0,C 180,E1 -24227.251,E2 -24227.251} C_VEL
LIN {X 0,Y 144.584,Z 513.385,A -85,B 0,C 180,E1 -24232.888,E2 -24232.888} C_VEL
LIN {X 0,Y 148.327,Z 507.632,A -85,B 0,C 180,E1 -24238.286,E2 -24238.286} C_VEL
LIN {X 0,Y 153.282,Z 500.366,A -85,B 0,C 180,E1 -24243.384,E2 -24243.384} C_VEL
LIN {X 0,Y 158.539,Z 492.744,A -85,B 0,C 180,E1 -24247.48,E2 -24247.48} C_VEL
LIN {X 0,Y 161.873,Z 488.284,A -85,B 0,C 180,E1 -24249.421,E2 -24249.421} C_VEL
LIN {X 0,Y 171.386,Z 485.635,A -85,B 0,C 180,E1 -24254.2,E2 -24254.2} C_VEL
LIN {X 0,Y 180.59,Z 482.697,A -85,B 0,C 180,E1 -24257.686,E2 -24257.686} C_VEL
LIN {X 0,Y 185.52,Z 480.944,A -85,B 0,C 180,E1 -24259.261,E2 -24259.261} C_VEL
LIN {X 0,Y 190.818,Z 479.008,A -85,B 0,C 180,E1 -24260.668,E2 -24260.668} C_VEL
LIN {X 0,Y 192.882,Z 477.925,A -85,B 0,C 180,E1 -24261.726,E2 -24261.726} C_VEL
LIN {X 0,Y 183.007,Z 478.21,A -85,B 0,C 180,E1 -24264.828,E2 -24264.828} C_VEL
LIN {X 0,Y 173.985,Z 477.337,A -85,B 0,C 180,E1 -24268.324,E2 -24268.324} C_VEL
LIN {X 0,Y 165.875,Z 475.26,A -85,B 0,C 180,E1 -24272.221,E2 -24272.221} C_VEL
LIN {X 0,Y 158.799,Z 471.938,A -85,B 0,C 180,E1 -24276.527,E2 -24276.527} C_VEL
LIN {X 0,Y 153.002,Z 467.315,A -85,B 0,C 180,E1 -24281.244,E2 -24281.244} C_VEL
LIN {X 0,Y 148.698,Z 461.302,A -85,B 0,C 180,E1 -24286.331,E2 -24286.331} C_VEL
LIN {X 0,Y 145.567,Z 453.752,A -85,B 0,C 180,E1 -24291.672,E2 -24291.672} C_VEL
LIN {X 0,Y 143.806,Z 445.71,A -85,B 0,C 180,E1 -24296.498,E2 -24296.498} C_VEL
LIN {X 0,Y 143.162,Z 435.565,A -85,B 0,C 180,E1 -24301.671,E2 -24301.671} C_VEL
LIN {X 0,Y 143.062,Z 435.638,A -85,B 0,C 180,E1 -24302.816,E2 -24302.816} C_VEL
LIN {X 0,Y 144.433,Z 433.821,A -85,B 0,C 180,E1 -24305.585,E2 -24305.585} C_VEL
LIN {X 0,Y 146.805,Z 430.919,A -85,B 0,C 180,E1 -24308.258,E2 -24308.258} C_VEL
LIN {X 0,Y 148.689,Z 429.191,A -85,B 0,C 180,E1 -24310.899,E2 -24310.899} C_VEL
LIN {X 0,Y 151.913,Z 425.768,A -85,B 0,C 180,E1 -24313.375,E2 -24313.375} C_VEL
LIN {X 0,Y 154.638,Z 423.607,A -85,B 0,C 180,E1 -24315.825,E2 -24315.825} C_VEL
LIN {X 0,Y 157.239,Z 421.181,A -85,B 0,C 180,E1 -24317.56,E2 -24317.56} C_VEL
LIN {X 0,Y 160.472,Z 417.911,A -85,B 0,C 180,E1 -24319.237,E2 -24319.237} C_VEL
LIN {X 0,Y 163.933,Z 415.3,A -85,B 0,C 180,E1 -24321.371,E2 -24321.371} C_VEL
LIN {X 0,Y 168.287,Z 410.897,A -85,B 0,C 180,E1 -24323.247,E2 -24323.247} C_VEL
LIN {X 0,Y 171.191,Z 407.665,A -85,B 0,C 180,E1 -24324.239,E2 -24324.239} C_VEL
LIN {X 0,Y 174.355,Z 404.964,A -85,B 0,C 180,E1 -24325.679,E2 -24325.679} C_VEL
LIN {X 0,Y 178.058,Z 401.196,A -85,B 0,C 180,E1 -24327.003,E2 -24327.003} C_VEL
LIN {X 0,Y 182.513,Z 395.783,A -85,B 0,C 180,E1 -24328.294,E2 -24328.294} C_VEL
LIN {X 0,Y 186.718,Z 389.838,A -85,B 0,C 180,E1 -24329.296,E2 -24329.296} C_VEL
LIN {X 0,Y 190.509,Z 385.56,A -85,B 0,C 180,E1 -24330.481,E2 -24330.481} C_VEL
LIN {X 0,Y 195.338,Z 378.769,A -85,B 0,C 180,E1 -24331.723,E2 -24331.723} C_VEL
LIN {X 0,Y 199.997,Z 370.529,A -85,B 0,C 180,E1 -24332.721,E2 -24332.721} C_VEL
LIN {X 0,Y 204.79,Z 359.304,A -85,B 0,C 180,E1 -24333.6,E2 -24333.6} C_VEL
LIN {X 0,Y 207.119,Z 352.531,A -85,B 0,C 180,E1 -24334.049,E2 -24334.049} C_VEL
LIN {X 0,Y 207.926,Z 351.337,A -85,B 0,C 180,E1 -24334.3,E2 -24334.3} C_VEL
LIN {X 0,Y 206.115,Z 366.909,A -85,B 0,C 180,E1 -24334.938,E2 -24334.938} C_VEL
LIN {X 0,Y 203.294,Z 382.375,A -85,B 0,C 180,E1 -24335.905,E2 -24335.905} C_VEL
LIN {X 0,Y 199.698,Z 397.163,A -85,B 0,C 180,E1 -24337.224,E2 -24337.224} C_VEL
LIN {X 0,Y 195.174,Z 411.421,A -85,B 0,C 180,E1 -24338.855,E2 -24338.855} C_VEL
LIN {X 0,Y 190.08,Z 424.364,A -85,B 0,C 180,E1 -24340.711,E2 -24340.711} C_VEL
LIN {X 0,Y 184.578,Z 436.272,A -85,B 0,C 180,E1 -24342.861,E2 -24342.861} C_VEL
LIN {X 0,Y 178.366,Z 448.126,A -85,B 0,C 180,E1 -24345.619,E2 -24345.619} C_VEL
LIN {X 0,Y 172.727,Z 458.034,A -85,B 0,C 180,E1 -24348.606,E2 -24348.606} C_VEL
LIN {X 0,Y 166.337,Z 467.725,A -85,B 0,C 180,E1 -24352.215,E2 -24352.215} C_VEL
LIN {X 0,Y 160.636,Z 475.715,A -85,B 0,C 180,E1 -24356.071,E2 -24356.071} C_VEL
LIN {X 0,Y 155.749,Z 482.346,A -85,B 0,C 180,E1 -24360.237,E2 -24360.237} C_VEL
LIN {X 0,Y 150.915,Z 488.456,A -85,B 0,C 180,E1 -24365.217,E2 -24365.217} C_VEL
LIN {X 0,Y 147.198,Z 493.157,A -85,B 0,C 180,E1 -24370.472,E2 -24370.472} C_VEL
LIN {X 0,Y 144.458,Z 496.593,A -85,B 0,C 180,E1 -24375.918,E2 -24375.918} C_VEL
LIN {X 0,Y 142.733,Z 498.847,A -85,B 0,C 180,E1 -24381.502,E2 -24381.502} C_VEL
LIN {X 0,Y 141.943,Z 499.983,A -85,B 0,C 180,E1 -24387.158,E2 -24387.158} C_VEL
LIN {X 0,Y 141.94,Z 499.992,A -85,B 0,C 180,E1 -24392.834,E2 -24392.834} C_VEL
LIN {X 0,Y 142.724,Z 498.895,A -85,B 0,C 180,E1 -24398.491,E2 -24398.491} C_VEL
LIN {X 0,Y 144.452,Z 496.683,A -85,B 0,C 180,E1 -24404.075,E2 -24404.075} C_VEL
LIN {X 0,Y 147.152,Z 493.299,A -85,B 0,C 180,E1 -24409.527,E2 -24409.527} C_VEL
LIN {X 0,Y 150.835,Z 488.649,A -85,B 0,C 180,E1 -24414.789,E2 -24414.789} C_VEL
LIN {X 0,Y 155.664,Z 482.583,A -85,B 0,C 180,E1 -24419.773,E2 -24419.773} C_VEL
LIN {X 0,Y 161.303,Z 474.948,A -85,B 0,C 180,E1 -24424.496,E2 -24424.496} C_VEL
LIN {X 0,Y 167.114,Z 466.767,A -85,B 0,C 180,E1 -24428.335,E2 -24428.335} C_VEL
LIN {X 0,Y 173.502,Z 456.885,A -85,B 0,C 180,E1 -24431.936,E2 -24431.936} C_VEL
LIN {X 0,Y 179.715,Z 445.944,A -85,B 0,C 180,E1 -24435.086,E2 -24435.086} C_VEL
LIN {X 0,Y 185.614,Z 434.617,A -85,B 0,C 180,E1 -24437.586,E2 -24437.586} C_VEL
LIN {X 0,Y 191.094,Z 422.407,A -85,B 0,C 180,E1 -24439.737,E2 -24439.737} C_VEL
LIN {X 0,Y 195.65,Z 410.682,A -85,B 0,C 180,E1 -24441.374,E2 -24441.374} C_VEL
LIN {X 0,Y 200.094,Z 396.513,A -85,B 0,C 180,E1 -24442.975,E2 -24442.975} C_VEL
LIN {X 0,Y 203.538,Z 382.276,A -85,B 0,C 180,E1 -24444.23,E2 -24444.23} C_VEL
LIN {X 0,Y 206.249,Z 367.285,A -85,B 0,C 180,E1 -24445.18,E2 -24445.18} C_VEL
LIN {X 0,Y 208.126,Z 351.55,A -85,B 0,C 180,E1 -24445.819,E2 -24445.819} C_VEL
LIN {X 0,Y 214.224,Z 276.558,A -85,B 0,C 180,E1 -24447.88,E2 -24447.88} C_VEL
LIN {X 0,Y 208.999,Z 265.767,A -85,B 0,C 180,E1 -24451.038,E2 -24451.038} C_VEL
LIN {X 0,Y 204.841,Z 258.169,A -85,B 0,C 180,E1 -24453.853,E2 -24453.853} C_VEL
LIN {X 0,Y 200.753,Z 251.357,A -85,B 0,C 180,E1 -24457.01,E2 -24457.01} C_VEL
LIN {X 0,Y 196.701,Z 245.024,A -85,B 0,C 180,E1 -24460.74,E2 -24460.74} C_VEL
LIN {X 0,Y 193.534,Z 240.532,A -85,B 0,C 180,E1 -24464.33,E2 -24464.33} C_VEL
LIN {X 0,Y 191.031,Z 236.825,A -85,B 0,C 180,E1 -24468.057,E2 -24468.057} C_VEL
LIN {X 0,Y 188.129,Z 232.68,A -85,B 0,C 180,E1 -24475.715,E2 -24475.715} C_VEL
LIN {X 0,Y 187.869,Z 232.02,A -85,B 0,C 180,E1 -24477.856,E2 -24477.856} C_VEL
LIN {X 0,Y 187.848,Z 232.048,A -85,B 0,C 180,E1 -24481.072,E2 -24481.072} C_VEL
LIN {X 0,Y 190.328,Z 236.838,A -85,B 0,C 180,E1 -24489.967,E2 -24489.967} C_VEL
LIN {X 0,Y 193.456,Z 241.764,A -85,B 0,C 180,E1 -24494.866,E2 -24494.866} C_VEL
LIN {X 0,Y 196.628,Z 246.695,A -85,B 0,C 180,E1 -24498.494,E2 -24498.494} C_VEL
LIN {X 0,Y 200.497,Z 252.944,A -85,B 0,C 180,E1 -24502.069,E2 -24502.069} C_VEL
LIN {X 0,Y 204.087,Z 259.037,A -85,B 0,C 180,E1 -24504.883,E2 -24504.883} C_VEL
LIN {X 0,Y 208.467,Z 267.002,A -85,B 0,C 180,E1 -24507.889,E2 -24507.889} C_VEL
LIN {X 0,Y 212.131,Z 280.981,A -85,B 0,C 180,E1 -24510.583,E2 -24510.583} C_VEL
LIN {X 0,Y 212.165,Z 298.442,A -85,B 0,C 180,E1 -24511.702,E2 -24511.702} C_VEL
LIN {X 0,Y 205.757,Z 375.506,A -85,B 0,C 180,E1 -24513.827,E2 -24513.827} C_VEL
LIN {X 0,Y 204.664,Z 381.312,A -85,B 0,C 180,E1 -24513.881,E2 -24513.881} C_VEL
LIN {X 0,Y 201.421,Z 390.652,A -85,B 0,C 180,E1 -24513.607,E2 -24513.607} C_VEL
LIN {X 0,Y 197.768,Z 399.898,A -85,B 0,C 180,E1 -24513.407,E2 -24513.407} C_VEL
LIN {X 0,Y 195.992,Z 405.457,A -85,B 0,C 180,E1 -24513.625,E2 -24513.625} C_VEL
LIN {X 0,Y 191.483,Z 420.185,A -85,B 0,C 180,E1 -24514.798,E2 -24514.798} C_VEL
LIN {X 0,Y 186.264,Z 433.892,A -85,B 0,C 180,E1 -24516.249,E2 -24516.249} C_VEL
LIN {X 0,Y 180.553,Z 446.501,A -85,B 0,C 180,E1 -24517.985,E2 -24517.985} C_VEL
LIN {X 0,Y 174.564,Z 458.22,A -85,B 0,C 180,E1 -24520.103,E2 -24520.103} C_VEL
LIN {X 0,Y 168.85,Z 468.219,A -85,B 0,C 180,E1 -24522.376,E2 -24522.376} C_VEL
LIN {X 0,Y 162.364,Z 478.439,A -85,B 0,C 180,E1 -24525.306,E2 -24525.306} C_VEL
LIN {X 0,Y 155.623,Z 488.455,A -85,B 0,C 180,E1 -24529.098,E2 -24529.098} C_VEL
LIN {X 0,Y 149.451,Z 496.863,A -85,B 0,C 180,E1 -24533.223,E2 -24533.223} C_VEL
LIN {X 0,Y 144.507,Z 503.731,A -85,B 0,C 180,E1 -24537.662,E2 -24537.662} C_VEL
LIN {X 0,Y 139.808,Z 510.194,A -85,B 0,C 180,E1 -24543.105,E2 -24543.105} C_VEL
LIN {X 0,Y 136.501,Z 515.233,A -85,B 0,C 180,E1 -24548.879,E2 -24548.879} C_VEL
LIN {X 0,Y 134.491,Z 518.96,A -85,B 0,C 180,E1 -24554.858,E2 -24554.858} C_VEL
LIN {X 0,Y 133.907,Z 521.475,A -85,B 0,C 180,E1 -24560.945,E2 -24560.945} C_VEL
LIN {X 0,Y 134.177,Z 522.365,A -85,B 0,C 180,E1 -24564.376,E2 -24564.376} C_VEL
LIN {X 0,Y 134.68,Z 522.987,A -85,B 0,C 180,E1 -24570.004,E2 -24570.004} C_VEL
LIN {X 0,Y 134.397,Z 522.794,A -85,B 0,C 180,E1 -24573.001,E2 -24573.001} C_VEL
LIN {X 0,Y 134.18,Z 522.283,A -85,B 0,C 180,E1 -24576.017,E2 -24576.017} C_VEL
LIN {X 0,Y 134.086,Z 520.336,A -85,B 0,C 180,E1 -24582.106,E2 -24582.106} C_VEL
LIN {X 0,Y 135.364,Z 517.195,A -85,B 0,C 180,E1 -24588.154,E2 -24588.154} C_VEL
LIN {X 0,Y 137.956,Z 512.788,A -85,B 0,C 180,E1 -24594.055,E2 -24594.055} C_VEL
LIN {X 0,Y 142.025,Z 507.036,A -85,B 0,C 180,E1 -24599.663,E2 -24599.663} C_VEL
LIN {X 0,Y 147.327,Z 499.771,A -85,B 0,C 180,E1 -24604.925,E2 -24604.925} C_VEL
LIN {X 0,Y 152.101,Z 493.236,A -85,B 0,C 180,E1 -24608.597,E2 -24608.597} C_VEL
LIN {X 0,Y 157.188,Z 486.841,A -85,B 0,C 180,E1 -24611.478,E2 -24611.478} C_VEL
LIN {X 0,Y 166.372,Z 484.776,A -85,B 0,C 180,E1 -24615.904,E2 -24615.904} C_VEL
LIN {X 0,Y 180.971,Z 480.682,A -85,B 0,C 180,E1 -24620.963,E2 -24620.963} C_VEL
LIN {X 0,Y 182.348,Z 479.93,A -85,B 0,C 180,E1 -24621.927,E2 -24621.927} C_VEL
LIN {X 0,Y 172.559,Z 479.174,A -85,B 0,C 180,E1 -24625.237,E2 -24625.237} C_VEL
LIN {X 0,Y 163.727,Z 477.24,A -85,B 0,C 180,E1 -24628.996,E2 -24628.996} C_VEL
LIN {X 0,Y 155.796,Z 474.112,A -85,B 0,C 180,E1 -24633.186,E2 -24633.186} C_VEL
LIN {X 0,Y 149.218,Z 469.725,A -85,B 0,C 180,E1 -24637.865,E2 -24637.865} C_VEL
LIN {X 0,Y 143.854,Z 464.007,A -85,B 0,C 180,E1 -24642.955,E2 -24642.955} C_VEL
LIN {X 0,Y 140.092,Z 456.801,A -85,B 0,C 180,E1 -24648.424,E2 -24648.424} C_VEL
LIN {X 0,Y 137.75,Z 449.125,A -85,B 0,C 180,E1 -24653.409,E2 -24653.409} C_VEL
LIN {X 0,Y 137.083,Z 445.705,A -85,B 0,C 180,E1 -24655.406,E2 -24655.406} C_VEL
LIN {X 0,Y 136.68,Z 445.57,A -85,B 0,C 180,E1 -24657.053,E2 -24657.053} C_VEL
LIN {X 0,Y 137.384,Z 443.827,A -85,B 0,C 180,E1 -24660,E2 -24660} C_VEL
LIN {X 0,Y 138.962,Z 441.406,A -85,B 0,C 180,E1 -24662.899,E2 -24662.899} C_VEL
LIN {X 0,Y 140.236,Z 439.849,A -85,B 0,C 180,E1 -24665.753,E2 -24665.753} C_VEL
LIN {X 0,Y 142.561,Z 437.236,A -85,B 0,C 180,E1 -24668.505,E2 -24668.505} C_VEL
LIN {X 0,Y 145.936,Z 434.24,A -85,B 0,C 180,E1 -24672.516,E2 -24672.516} C_VEL
LIN {X 0,Y 149.392,Z 431.007,A -85,B 0,C 180,E1 -24674.996,E2 -24674.996} C_VEL
LIN {X 0,Y 152.382,Z 428.77,A -85,B 0,C 180,E1 -24677.445,E2 -24677.445} C_VEL
LIN {X 0,Y 154.174,Z 427.301,A -85,B 0,C 180,E1 -24678.608,E2 -24678.608} C_VEL
LIN {X 0,Y 158.548,Z 423.331,A -85,B 0,C 180,E1 -24680.77,E2 -24680.77} C_VEL
LIN {X 0,Y 162.341,Z 420.603,A -85,B 0,C 180,E1 -24682.931,E2 -24682.931} C_VEL
LIN {X 0,Y 167.207,Z 416.13,A -85,B 0,C 180,E1 -24684.855,E2 -24684.855} C_VEL
LIN {X 0,Y 169.927,Z 413.366,A -85,B 0,C 180,E1 -24685.739,E2 -24685.739} C_VEL
LIN {X 0,Y 175.661,Z 408.435,A -85,B 0,C 180,E1 -24687.913,E2 -24687.913} C_VEL
LIN {X 0,Y 180.713,Z 403.2,A -85,B 0,C 180,E1 -24689.39,E2 -24689.39} C_VEL
LIN {X 0,Y 186.146,Z 396.506,A -85,B 0,C 180,E1 -24690.644,E2 -24690.644} C_VEL
LIN {X 0,Y 187.732,Z 394.362,A -85,B 0,C 180,E1 -24690.981,E2 -24690.981} C_VEL
LIN {X 0,Y 191.803,Z 389.987,A -85,B 0,C 180,E1 -24692.093,E2 -24692.093} C_VEL
LIN {X 0,Y 197.015,Z 383.143,A -85,B 0,C 180,E1 -24693.28,E2 -24693.28} C_VEL
LIN {X 0,Y 200.199,Z 378.11,A -85,B 0,C 180,E1 -24693.914,E2 -24693.914} C_VEL
LIN {X 0,Y 196.932,Z 392.388,A -85,B 0,C 180,E1 -24695.053,E2 -24695.053} C_VEL
LIN {X 0,Y 192.584,Z 406.982,A -85,B 0,C 180,E1 -24696.593,E2 -24696.593} C_VEL
LIN {X 0,Y 187.841,Z 419.481,A -85,B 0,C 180,E1 -24698.21,E2 -24698.21} C_VEL
LIN {X 0,Y 182.144,Z 432.297,A -85,B 0,C 180,E1 -24700.351,E2 -24700.351} C_VEL
LIN {X 0,Y 176.268,Z 443.519,A -85,B 0,C 180,E1 -24702.673,E2 -24702.673} C_VEL
LIN {X 0,Y 170.389,Z 453.878,A -85,B 0,C 180,E1 -24705.473,E2 -24705.473} C_VEL
LIN {X 0,Y 164.513,Z 462.979,A -85,B 0,C 180,E1 -24708.531,E2 -24708.531} C_VEL
LIN {X 0,Y 158.133,Z 471.913,A -85,B 0,C 180,E1 -24712.327,E2 -24712.327} C_VEL
LIN {X 0,Y 152.483,Z 479.304,A -85,B 0,C 180,E1 -24716.417,E2 -24716.417} C_VEL
LIN {X 0,Y 148.229,Z 484.617,A -85,B 0,C 180,E1 -24720.139,E2 -24720.139} C_VEL
LIN {X 0,Y 143.406,Z 490.364,A -85,B 0,C 180,E1 -24725.378,E2 -24725.378} C_VEL
LIN {X 0,Y 140.522,Z 493.744,A -85,B 0,C 180,E1 -24729.503,E2 -24729.503} C_VEL
LIN {X 0,Y 137.614,Z 497.177,A -85,B 0,C 180,E1 -24735.202,E2 -24735.202} C_VEL
LIN {X 0,Y 135.75,Z 499.431,A -85,B 0,C 180,E1 -24741.061,E2 -24741.061} C_VEL
LIN {X 0,Y 134.874,Z 500.568,A -85,B 0,C 180,E1 -24747.009,E2 -24747.009} C_VEL
LIN {X 0,Y 134.871,Z 500.577,A -85,B 0,C 180,E1 -24752.983,E2 -24752.983} C_VEL
LIN {X 0,Y 135.741,Z 499.479,A -85,B 0,C 180,E1 -24758.932,E2 -24758.932} C_VEL
LIN {X 0,Y 137.606,Z 497.266,A -85,B 0,C 180,E1 -24764.791,E2 -24764.791} C_VEL
LIN {X 0,Y 140.477,Z 493.885,A -85,B 0,C 180,E1 -24770.496,E2 -24770.496} C_VEL
LIN {X 0,Y 144.422,Z 489.234,A -85,B 0,C 180,E1 -24775.97,E2 -24775.97} C_VEL
LIN {X 0,Y 149.555,Z 483.165,A -85,B 0,C 180,E1 -24781.122,E2 -24781.122} C_VEL
LIN {X 0,Y 155.506,Z 475.53,A -85,B 0,C 180,E1 -24785.977,E2 -24785.977} C_VEL
LIN {X 0,Y 161.623,Z 467.346,A -85,B 0,C 180,E1 -24789.891,E2 -24789.891} C_VEL
LIN {X 0,Y 168.288,Z 457.464,A -85,B 0,C 180,E1 -24793.552,E2 -24793.552} C_VEL
LIN {X 0,Y 174.332,Z 447.354,A -85,B 0,C 180,E1 -24796.518,E2 -24796.518} C_VEL
LIN {X 0,Y 180.363,Z 436.33,A -85,B 0,C 180,E1 -24799.017,E2 -24799.017} C_VEL
LIN {X 0,Y 186.047,Z 424.337,A -85,B 0,C 180,E1 -24801.175,E2 -24801.175} C_VEL
LIN {X 0,Y 191.324,Z 411.245,A -85,B 0,C 180,E1 -24803.025,E2 -24803.025} C_VEL
LIN {X 0,Y 195.838,Z 397.354,A -85,B 0,C 180,E1 -24804.595,E2 -24804.595} C_VEL
LIN {X 0,Y 199.586,Z 382.411,A -85,B 0,C 180,E1 -24805.905,E2 -24805.905} C_VEL
LIN {X 0,Y 202.422,Z 366.976,A -85,B 0,C 180,E1 -24806.864,E2 -24806.864} C_VEL
LIN {X 0,Y 204.278,Z 351.513,A -85,B 0,C 180,E1 -24807.475,E2 -24807.475} C_VEL
